(* IEC 61131-3 sources: elnaProjects/kc6/build_BaseProject_ecl/_ (part 3) *)

  StrAlg.status :=  SHL(BYTE_TO_DWORD(source_for_Status), 29)
  			OR SHL(BYTE_TO_DWORD(cmd_for_Status), 26)
  			OR SHL(BYTE_TO_DWORD(command_error_for_Status), 23)
  			OR SHL(BOOL_TO_DWORD(StrAlg.OpcCommandsDisabled ), 21)
  			OR SHL(BOOL_TO_DWORD(StrAlg.hasError),4)
  			OR SHL(BOOL_TO_DWORD(StrAlg.CanRun),2)
  			OR SHL(BOOL_TO_DWORD(StrAlg.isEnded),1)
  			OR BOOL_TO_DWORD(StrAlg.isRuning);
END_FUNCTION_BLOCK

FUNCTION_BLOCK TestProtectionAlg
  VAR_IN_OUT
    StrAlg : struct_Alg;
  END_VAR
  VAR
    _sunpackerCommand : fb_sunpackerCommand;
    source : BYTE;
    cmd : BYTE;
    lastCmd : BYTE;
    source_for_Status : BYTE;
    cmd_for_Status : BYTE;
    command_error_for_Status : BYTE;
    resetCmdTimer : TON;
    resetCmdTimerPriznak : BOOL;
  END_VAR
  VAR_EXTERNAL
    ai : AiConfig;
    protectManager : struct_ProtectionsManager;
    algManager : struct_AlgoritmsManager;
    ModeGpa : TYPE_ModeGpa;
    PMcommand : TYPE_CommandsPotectionsManager;
  END_VAR

  StrAlg.CanRun := StrAlg.inCanRun;
  StrAlg.OpcCommandsDisabled := StrAlg.inOpcCommandsDisabled;

  (* ---- Если управление с ВУ заблокировано, то передаем команду из алгоритма ---- *)
  IF StrAlg.inOpcCommandsDisabled THEN
  	StrAlg.inCommand := StrAlg.inCommand_Alg;
  ELSE (* иначе передаем команду с АРМа*)
  	StrAlg.inCommand := StrAlg.inCommand_ARM;
  END_IF;

  _sunpackerCommand(command := StrAlg.inCommand);
  	source := _sunpackerCommand.source;
  	cmd := _sunpackerCommand.cmd;

  IF cmd <> 0 AND lastCmd <> cmd AND (((NOT StrAlg.opcCommandsDisabled) AND source > 0) OR source = 0) then
  	CASE BYTE_TO_INT(cmd) OF
  		(*cmdRun*) 1: 	IF (StrAlg.CanRun) THEN
  					StrAlg.isRuning := TRUE;
  					StrAlg.isEnded := FALSE;
  					StrAlg.hasError 	:= FALSE;
                                               (*****************       OnRun       *****************)
                                                        algManager.nMode:=ModeGpa.MODE_TESTAZ;
                                                        protectManager.inCommand:=PMcommand.CheckProtections;
  					    EnableAiLimits(ai);
                                                    (*StrAlg.inOpcCommandsDisabled:=FALSE;*)
  					cmd_for_Status := cmd;
  					source_for_Status := source;
  					command_error_for_Status := 0;
  				ELSE
  					StrAlg.isRuning := FALSE;
  					StrAlg.isEnded := FALSE;
  					StrAlg.hasError 	:= FALSE;

  					cmd_for_Status := 0;
  					source_for_Status := source;
  					command_error_for_Status := cmd;
  				END_IF;
  		(*cmdReset*) 2: 	StrAlg.isRuning := FALSE;
  				StrAlg.isEnded := FALSE;
  				StrAlg.hasError 	:= FALSE;
                                          (*****************       OnReset       *****************)
                                                    DisableAiLimits(ai);
                                                    protectManager.inCommand:=PMcommand.RestartAllProtections;
                                                    algManager.nMode:=ModeGpa.MODE_STOP;

  				cmd_for_Status := cmd;
  				source_for_Status := source;
  				command_error_for_Status := 0;
  	END_CASE;
  	resetCmdTimer(IN := false);
  	resetCmdTimerPriznak := TRUE;
  END_IF;
  lastCmd := cmd;

  resetCmdTimer(IN := resetCmdTimerPriznak, PT := T#5S);
  IF resetCmdTimer.Q THEN
  	resetCmdTimerPriznak := FALSE;
  	source_for_Status := 0;
  	cmd_for_Status := 0;
  	command_error_for_Status := 0;
  END_IF;

  StrAlg.status :=  SHL(BYTE_TO_DWORD(source_for_Status), 29)
  			OR SHL(BYTE_TO_DWORD(cmd_for_Status), 26)
  			OR SHL(BYTE_TO_DWORD(command_error_for_Status), 23)
  			OR SHL(BOOL_TO_DWORD(StrAlg.OpcCommandsDisabled ), 21)
  			OR SHL(BOOL_TO_DWORD(StrAlg.hasError),4)
  			OR SHL(BOOL_TO_DWORD(StrAlg.CanRun),2)
  			OR SHL(BOOL_TO_DWORD(StrAlg.isEnded),1)
  			OR BOOL_TO_DWORD(StrAlg.isRuning);
END_FUNCTION_BLOCK

FUNCTION_BLOCK engineRunAlg
  VAR_IN_OUT
    StrAlg : struct_Alg;
  END_VAR
  VAR
    BreakPuskTimer : struct_PhaseAlgoritm;
    RunProtection_mvoff : struct_PhaseAlgoritm;
    LowOil_upStopust : struct_PhaseAlgoritm;
    mvOn : struct_PhaseAlgoritm;
    AutoPns_ph : struct_PhaseAlgoritm;
    AutoAvom_ph : struct_PhaseAlgoritm;
    pnsOff : struct_PhaseAlgoritm;
    testUnsuccessful : struct_PhaseAlgoritm;
    fb_BreakPuskTimer : fb_ph_Timer;
    fb_RunProtection_mvoff : fb_ph_DIprotection;
    fb_LowOil_upStopust : fb_ph_WaitAnalogValue;
    fb_mvOn : fb_ph_SectionSwitch;
    fb_AutoPns_ph : fb_ph_algoritm;
    fb_AutoAvom_ph : fb_ph_algoritm;
    fb_pnsOff : fb_ph_Switch;
    fb_testUnsuccessful : fb_ph_CustomPhase;
    _sunpackerCommand : fb_sunpackerCommand;
    _DualStateImAction : TYPE_DualStateImAction;
    _PhaseAlgoritmAction : TYPE_PhaseAlgoritmAction;
    source : BYTE;
    cmd : BYTE;
    lastCmd : BYTE;
    source_for_Status : BYTE;
    cmd_for_Status : BYTE;
    command_error_for_Status : BYTE;
    resetCmdTimer : TON;
    resetCmdTimerPriznak : BOOL;
    onInit : BOOL;
    waitReset : TON;
  END_VAR
  VAR_EXTERNAL
    IM : ImConfig;
    algoritms : AlgoritmsConfig;
    ai : AiConfig;
    protections : ProtectionsConfig;
    AlgTimers : struct_AlgTimers;
  END_VAR

  IF NOT onInit THEN

       fb_BreakPuskTimer(phaseNumber:=0, delay:=T#665S);
     fb_LowOil_upStopust(phaseNumber:=1);
                 fb_mvOn(phaseNumber:=2, act:=_on);
           fb_AutoPns_ph(phaseNumber:=3, act:=_run, waitCompletion:=FALSE);
          fb_AutoAvom_ph(phaseNumber:=4, act:=_run, waitCompletion:=FALSE);
               fb_pnsOff(phaseNumber:=5, act:=_off);
  fb_RunProtection_mvoff(phaseNumber:=7, act:=_run);
     fb_testUnsuccessful(phaseNumber:=17);

  onInit:=TRUE;
  END_IF;

          fb_BreakPuskTimer(StrPh:=BreakPuskTimer, timer:=AlgTimers.engineRun_BreakPuskTimer);
        fb_LowOil_upStopust(StrPh:=LowOil_upStopust, ai:=ai.Davlenie_masla_smazki_nizkoe, more:=im.AutoPns_UstStop.Value);
                    fb_mvOn(StrPh:=mvOn, Im:=Im.MB);
              fb_AutoPns_ph(StrPh:=AutoPns_ph, alg:=algoritms.AutoPns);
             fb_AutoAvom_ph(StrPh:=AutoAvom_ph, alg:=algoritms.AutoAvom);
                  fb_pnsOff(StrPh:=pnsOff, Im:=Im.pns);
     fb_RunProtection_mvoff(StrPh:=RunProtection_mvoff, StrDiP:=protections.MB);
        fb_testUnsuccessful(StrPh:=testUnsuccessful);

  StrAlg.CanRun := StrAlg.inCanRun;
  StrAlg.OpcCommandsDisabled := StrAlg.inOpcCommandsDisabled;

  IF StrAlg.isRuning THEN

      StrAlg.hasError := mvOn.error OR pnsOff.error OR testUnsuccessful.error;

      IF mvOn.top THEN
          runPhase(RunProtection_mvoff);
          runPhase(AutoAvom_ph);
          runPhase(LowOil_upStopust);
      END_IF;

      IF LowOil_upStopust.top THEN
          runPhase(pnsOff);
      END_IF;

      IF pnsOff.top THEN
         runPhase(AutoPns_ph);
      END_IF;

      IF BreakPuskTimer.top AND NOT AutoPns_ph.top THEN
            testUnsuccessful.error:=TRUE;
      END_IF;

      IF AutoPns_ph.top THEN
            resetPhase(BreakPuskTimer);
  	waitReset(IN:=TRUE, PT:= T#2S);
      END_IF;

      IF waitReset.Q AND NOT (algoritms.Apusk.isRuning OR algoritms.SemiAutoPusk.isRuning) THEN
  	resetIfRunning(StrAlg);
      END_IF;

      StrAlg.isEnded:= AutoPns_ph.top;
  END_IF;

  StrAlg.CanRun := StrAlg.inCanRun;
  StrAlg.OpcCommandsDisabled := StrAlg.inOpcCommandsDisabled;

  (* ---- Если управление с ВУ заблокировано, то  передаем команду из алгоритма ---- *)
  IF StrAlg.inOpcCommandsDisabled THEN
  	StrAlg.inCommand := StrAlg.inCommand_Alg;
  ELSE (* иначе передаем команду с АРМа*)
  	StrAlg.inCommand := StrAlg.inCommand_ARM;
  END_IF;

  _sunpackerCommand(command := StrAlg.inCommand);
  	source := _sunpackerCommand.source;
  	cmd := _sunpackerCommand.cmd;

  IF cmd <> 0 AND lastCmd <> cmd AND (((NOT StrAlg.opcCommandsDisabled) AND source > 0) OR source = 0) then
  	CASE BYTE_TO_INT(cmd) OF
  		(*cmdRun*) 1: 	IF (StrAlg.CanRun) THEN
  					StrAlg.isRuning := TRUE;
  					StrAlg.isEnded := FALSE;
  					StrAlg.hasError := FALSE;
  					(*****************       OnRun       *****************)

                                                    runPhase(mvOn);
                                                    runPhase(BreakPuskTimer);
                                                    runPhase(testUnsuccessful);

  					cmd_for_Status := cmd;
  					source_for_Status := source;
  					command_error_for_Status := 0;
  				ELSE
  					StrAlg.isRuning := FALSE;
  					StrAlg.isEnded := FALSE;
  					StrAlg.hasError 	:= FALSE;

  					cmd_for_Status := 0;
  					source_for_Status := source;
  					command_error_for_Status := cmd;
  				END_IF;
  		(*cmdReset*) 2: 	StrAlg.isRuning := FALSE;
  				StrAlg.isEnded := FALSE;
  				StrAlg.hasError 	:= FALSE;

                                           (*****************       OnReset       *****************)
                                          StrAlg.inCanRun:=FALSE;
                                          waitReset(IN:=FALSE);

                                          resetPhase(BreakPuskTimer);
                                          resetPhase(RunProtection_mvoff);
                                          resetPhase(LowOil_upStopust);
                                          resetPhase(mvOn);
                                          resetPhase(AutoPns_ph);
                                          resetPhase(AutoAvom_ph);
                                          resetPhase(pnsOff);
                                          resetPhase(testUnsuccessful);

  				cmd_for_Status := cmd;
  				source_for_Status := source;
  				command_error_for_Status := 0;
  	END_CASE;
  	resetCmdTimer(IN := false);
  	resetCmdTimerPriznak := TRUE;
  END_IF;
  lastCmd := cmd;

  resetCmdTimer(IN := resetCmdTimerPriznak, PT := T#5S);
  IF resetCmdTimer.Q THEN
  	resetCmdTimerPriznak := FALSE;
  	source_for_Status := 0;
  	cmd_for_Status := 0;
  	command_error_for_Status := 0;
  END_IF;

  StrAlg.Start:= BreakPuskTimer.startStatus
              OR RunProtection_mvoff.startStatus
              OR LowOil_upStopust.startStatus
              OR mvOn.startStatus
              OR AutoPns_ph.startStatus
              OR AutoAvom_ph.startStatus
              OR pnsOff.startStatus
              OR testUnsuccessful.startStatus;

  StrAlg.Error:= BreakPuskTimer.errorStatus
              OR RunProtection_mvoff.errorStatus
              OR LowOil_upStopust.errorStatus
              OR mvOn.errorStatus
              OR AutoPns_ph.errorStatus
              OR AutoAvom_ph.errorStatus
              OR pnsOff.errorStatus
              OR testUnsuccessful.errorStatus;

  StrAlg.Top:=   BreakPuskTimer.topStatus
              OR RunProtection_mvoff.topStatus
              OR LowOil_upStopust.topStatus
              OR mvOn.topStatus
              OR AutoPns_ph.topStatus
              OR AutoAvom_ph.topStatus
              OR pnsOff.topStatus
              OR testUnsuccessful.topStatus;

  (*TODO: TYPE PROGRAM CODE HERE*)
  StrAlg.status :=  SHL(BYTE_TO_DWORD(source_for_Status), 29)
  			OR SHL(BYTE_TO_DWORD(cmd_for_Status), 26)
  			OR SHL(BYTE_TO_DWORD(command_error_for_Status), 23)
  			OR SHL(BOOL_TO_DWORD(StrAlg.OpcCommandsDisabled ), 21)
  			OR SHL(BOOL_TO_DWORD(StrAlg.hasError),4)
  			OR SHL(BOOL_TO_DWORD(StrAlg.CanRun),2)
  			OR SHL(BOOL_TO_DWORD(StrAlg.isEnded),1)
  			OR BOOL_TO_DWORD(StrAlg.isRuning);
END_FUNCTION_BLOCK

FUNCTION_BLOCK fb_AI_Init
  VAR_INPUT
    data_Ini : BOOL;
    dLL : LREAL;
    dHL : LREAL;
    dLA : LREAL;
    dHA : LREAL;
    dLW : LREAL;
    dHW : LREAL;
    ISVALIDREF_LA : BOOL         := False;
    ISVALIDREF_HA : BOOL         := False;
    ISVALIDREF_LW : BOOL         := False;
    ISVALIDREF_HW : BOOL         := False;
    delayLA : TIME         := T#0S;
    delayLW : TIME         := T#0S;
    delayHW : TIME         := T#0S;
    delayHA : TIME         := T#0S;
    inpLL : LREAL         := 4000.0;
    inpHL : LREAL         := 20000.0;
    CurrentShotCircuit : LREAL         := 21000.0;
    CurrentBreakCircuit : LREAL         := 3700.0;
    dMaxChangeSpeed : LREAL;
    dMaxChangeSpeedDown : LREAL;
    histeresis : LREAL;
    aperturFilter : LREAL;
    exponentialFilter : LREAL;
    rassoglasovanie : LREAL;
    inOpcCommandsDisabled : BOOL;
  END_VAR
  VAR_IN_OUT
    strAI : struct_AI;
  END_VAR
  VAR_OUTPUT
    Init : BOOL         := FALSE;
  END_VAR

  (*****            Функциональный блок переинициализации структуры-дескриптора канала аналогового ввода.            *****)
       Init := false;

      IF data_Ini THEN                            (* Параметрам требуется переинициализация. *)
          strAI.dLL                := dLL;
          strAI.dHL                := dHL;
          strAI.dLA                := dLA;
          strAI.dHA                := dHA;
          strAI.dLW                := dLW;
          strAI.dHW                := dHW;
          strAI.ISVALIDREF_LA      := ISVALIDREF_LA;
          strAI.ISVALIDREF_HA      := ISVALIDREF_HA;
          strAI.ISVALIDREF_LW      := ISVALIDREF_LW;
          strAI.ISVALIDREF_HW      := ISVALIDREF_HW;
          strAI.delayLA            := delayLA;
          strAI.delayLW            := delayLW;
          strAI.delayHW            := delayHW;
          strAI.delayHA            := delayHA;
          strAI.inpLL              := inpLL;
          strAI.inpHL              := inpHL;
          strAI.CurrentShotCircuit := CurrentShotCircuit;
          strAI.CurrentBreakCircuit:= CurrentBreakCircuit;
          strAI.dMaxChangeSpeed     := dMaxChangeSpeed;
          strAI.dMaxChangeSpeedDown := dMaxChangeSpeedDown;
          strAI.histeresis         := histeresis;
          strAI.aperturFilter      := aperturFilter;
          strAI.exponentialFilter  := exponentialFilter;
          strAI.rassoglasovanie    := rassoglasovanie;
          strAI.rassoglasovanie    := rassoglasovanie;

          data_Ini:=false;
          Init := TRUE;
       END_IF;
    IF Init THEN
          dLL:= 0.0;
          dHL:= 0.0;
          dLA:= 0.0;
          dHA:= 0.0;
          dLW:= 0.0;
          dHW:= 0.0;
          inpLL:= 4000.0;
          inpHL:= 20000.0;
          CurrentShotCircuit:= 21000.0;
          CurrentBreakCircuit:= 3700.0;
          ISVALIDREF_LA:= false;
          ISVALIDREF_HA:= false;
          ISVALIDREF_LW:= false;
          ISVALIDREF_HW:= false;
          delayLA:= T#0S;
          delayLW:= T#0S;
          delayHW:= T#0S;
          delayHA:= T#0S;
          dMaxChangeSpeed:= 0.0;
          dMaxChangeSpeedDown:= 0.0;
          histeresis:= 0.0;
          aperturFilter:= 0.0;
          exponentialFilter:= 0.0;
          rassoglasovanie:= 0.0;
        END_IF;
END_FUNCTION_BLOCK

FUNCTION_BLOCK fb_AOSourceMlp
  VAR_IN_OUT
    OutCurrent : TDoubleData;
    strAO : struct_AO;
  END_VAR
  VAR_INPUT
    retainLL : LREAL;
    retainHL : LREAL;
  END_VAR
  VAR
    _sunpackerCommand : fb_sunpackerCommand;
    source : BYTE;
    source_for_Status : BYTE;
    cmd : BYTE;
    cmd_for_Status : BYTE;
    lastCmd : BYTE;
    command_error_for_Status : BYTE;
    resetCmdTimer : TON;
    resetCmdTimerPriznak : BOOL;
    secondTack : BOOL;
    inOpcCommandsDisabled : BOOL;
  END_VAR

  IF NOT secondTack THEN
            IF (strAO.newLL <> retainLL) AND (retainLL <> 0.0) THEN  strAO.LL := retainLL;
            ELSE strAO.LL:= strAO.newLL; END_IF;
  	IF (strAO.newHL <> retainHL) AND (retainHL <> 0.0) THEN  strAO.HL := retainHL;
            ELSE strAO.HL:= strAO.newHL; END_IF;

  	secondTack  := FALSE;
  END_IF;
  strAO.blConnect :=(UINT_TO_WORD(OutCurrent.wFlags) AND 16#0040) <> 0;
  strAO.OpcCommandsDisabled := inOpcCommandsDisabled;

  _sunpackerCommand(command := strAO.inCommand);
  	source := _sunpackerCommand.source;
  	cmd := _sunpackerCommand.cmd;

  IF cmd <> 0 AND lastCmd <> cmd and (((NOT strAO.opcCommandsDisabled) AND source > 0) OR source = 0) then
  	CASE BYTE_TO_INT(cmd) OF
  	(*cmd_ChangeValue*) 1 : 	IF ((NOT strAO.newLL_ISVALIDREF) OR (strAO.nValue >= strAO.LL)) AND
                                             ((NOT strAO.newHL_ISVALIDREF) OR (strAO.nValue <= strAO.HL) ) THEN
  					strAO.Value := strAO.nValue;
  				END_IF;
  	(*cmd_ChangeLimits*) 2 : 	strAO.LL := strAO.newLL; retainLL:= strAO.LL;
  				strAO.HL := strAO.newHL; retainHL:= strAO.HL;
  	END_CASE;
  	source_for_Status := source;
  	cmd_for_Status := cmd;
  	command_error_for_Status := 0;
  	resetCmdTimer(IN := FALSE);
  	resetCmdTimerPriznak := TRUE;
  END_IF;
  lastCmd := cmd;

  IF (strAO.HL <> strAO.LL) THEN
  	OutCurrent.dblValue := ((strAO.Value - strAO.LL) * (strAO.outHL-strAO.outLL)/(strAO.HL - strAO.LL )) + strAO.outLL;
  END_IF;

  resetCmdTimer(IN := resetCmdTimerPriznak, PT := T#5S);
  IF resetCmdTimer.Q THEN
  	resetCmdTimerPriznak := FALSE;
  	source_for_Status := 0;
  	cmd_for_Status := 0;
  	command_error_for_Status := 0;
  END_IF;

  strAO.status := SHL(BYTE_TO_DWORD(source_for_Status), 29)
  			OR SHL(BYTE_TO_DWORD(cmd_for_Status), 26)
  			OR SHL(BYTE_TO_DWORD(command_error_for_Status), 23)
  			OR SHL(BOOL_TO_DWORD(strAO.OpcCommandsDisabled ), 21);
END_FUNCTION_BLOCK

FUNCTION_BLOCK fb_AO_Init
  VAR_INPUT
    data_Ini : BOOL;
    outLL : LREAL         := 4000.0;
    outHL : LREAL         := 20000.0;
    newLL : LREAL;
    newHL : LREAL;
    newLL_ISVALIDREF : BOOL;
    newHL_ISVALIDREF : BOOL;
  END_VAR
  VAR_IN_OUT
    strAO : struct_AO;
  END_VAR
  VAR_OUTPUT
    Init : BOOL         := FALSE;
  END_VAR

  (*****            Функциональный блок переинициализации структуры-дескриптора канала аналогового ввода.            *****)

   Init := FALSE;

      IF data_Ini THEN                            (* Параметрам требуется переинициализация. *)
          strAO.outLL                := outLL;
          strAO.outHL                := outHL;
          strAO.newLL                := newLL;
          strAO.newHL                := newHL;
          strAO.newLL_ISVALIDREF     := newLL_ISVALIDREF;
          strAO.newHL_ISVALIDREF     := newHL_ISVALIDREF;
          data_Ini:=FALSE;
          Init := TRUE;
      END_IF;
   IF Init THEN
         (* outLL:=0.0;*)
         (* outHL:=0.0;*)
          newLL:=0.0;
          newHL:=0.0;
          newLL_ISVALIDREF:= FALSE;
          newHL_ISVALIDREF:= FALSE;
   END_IF;
END_FUNCTION_BLOCK

FUNCTION_BLOCK fb_AiProtection
  VAR_INPUT
    ai : struct_AI;
  END_VAR
  VAR_IN_OUT
    StrAIp : struct_AiProtection;
  END_VAR
  VAR
    _sunpackerCommand : fb_sunpackerCommand;
    _signalingTp : TOF;
    _statusAi : TYPE_StatusAi;
    source : BYTE;
    cmd : BYTE;
    lastCmd : BYTE;
    source_for_Status : BYTE;
    cmd_for_Status : BYTE;
    command_error_for_Status : BYTE;
    resetCmdTimer : TON;
    resetCmdTimerPriznak : BOOL;
    signalinTimer : TON;
    timer : TON;
    SignalingTrig : R_TRIG;
    SignalingFTrig : F_TRIG;
    SignalingAi : BOOL;
  END_VAR

  timer(IN :=(ai.interval=StrAIp.controlLimit) AND (ai.interval >= _statusAi.normal) AND StrAIp.isRunning, PT :=StrAIp.delay);
  SignalingTrig(CLK := timer.Q);
  IF SignalingTrig.Q THEN
  	SignalingAi := TRUE;
  END_IF;
  SignalingFTrig(CLK := timer.Q);
  IF SignalingFTrig.Q THEN
  	SignalingAi := FALSE;
  END_IF;

  StrAIp.Tag := StrAIp.inTag;
  StrAIp.RunOnStart := StrAIp.inRunOnStart;

  StrAIp.CanRun := StrAIp.inCanRun;

  StrAIp.OpcCommandsDisabled := StrAIp.inOpcCommandsDisabled;

  (* ---- Если управление с ВУ заблокировано, то передаем команду из алгоритма ---- *)
  IF StrAIp.inOpcCommandsDisabled THEN
  	StrAIp.inCommand := StrAIp.inCommand_Alg;
  ELSE (* иначе передаем команду с АРМа*)
  	StrAIp.inCommand := StrAIp.inCommand_ARM;
  END_IF;

  _sunpackerCommand(command := StrAIp.inCommand);
  	source := _sunpackerCommand.source;
  	cmd := _sunpackerCommand.cmd;

  IF cmd <> 0 AND lastCmd <> cmd AND (((NOT StrAIp.opcCommandsDisabled) AND source > 0) OR source = 0) then

  	CASE BYTE_TO_INT(cmd) OF
  		(*cmdRun*) 1: 	IF        NOT StrAIp.Remont THEN
  					StrAIp.isEnded := FALSE;
  					StrAIp.hasError 	:= FALSE;
  					StrAIp.isRunning := TRUE;

  					cmd_for_Status := cmd;
  					source_for_Status := source;
  					command_error_for_Status := 0;
  				ELSE
  					StrAIp.isRunning := FALSE;
  					StrAIp.isEnded := FALSE;
  					StrAIp.hasError 	:= FALSE;

  					cmd_for_Status := 0;
  					source_for_Status := source;
  					command_error_for_Status := cmd;
  				END_IF;
                                          StrAIp.inopcCommandsDisabled:=FALSE;

  		(*cmdReset*) 2: 	StrAIp.isRunning := FALSE;
  				StrAIp.isEnded := FALSE;
  				StrAIp.hasError 	:= FALSE;
  				SignalingAi := FALSE;
  				StrAIp.Check := FALSE;
                                          (*StrAIp.Remont := FALSE;*)
  				cmd_for_Status := cmd;
  				source_for_Status := source;
  				command_error_for_Status := 0;
                                          StrAIp.inopcCommandsDisabled:=FALSE;

  	(*cmd_setRemont*) 4 :	StrAIp.Remont := TRUE;
  				(*StrAIp.isRunning := FALSE;*)

  				cmd_for_Status := cmd;
  				source_for_Status := source;
  				command_error_for_Status := 0;
  	(*cmd_resetRemont*) 5 : 	(*IF (ai.interval=StrAIp.controlLimit) THEN
  					cmd_for_Status := 0;
  					source_for_Status := 0;
  					command_error_for_Status := cmd;
  				ELSE*)
  					StrAIp.Remont := FALSE;
  					(*StrAIp.isRunning := TRUE;*)

  					cmd_for_Status := cmd;
  					source_for_Status := source;
  					command_error_for_Status := 0;
  				(*END_IF;*)
  	(*cmd_setCheck*) 6 : 	StrAIp.Check := TRUE;

  				cmd_for_Status := cmd;
  				source_for_Status := source;
  				command_error_for_Status := 0;
  	END_CASE;
  	resetCmdTimer(IN := false);
  	resetCmdTimerPriznak := TRUE;
  END_IF;
  lastCmd := cmd;

  resetCmdTimer(IN := resetCmdTimerPriznak);
  IF resetCmdTimer.Q THEN
  	resetCmdTimerPriznak := FALSE;
  	source_for_Status := 0;
  	cmd_for_Status := 0;
  	command_error_for_Status := 0;
  END_IF;

  IF StrAIp.isRunning AND NOT StrAIp.Remont AND NOT StrAIp.Check THEN
  	StrAIp.Signaling := SignalingAi;
  	StrAIp.SignalingTP := _signalingTp.Q;
  ELSE
  	StrAIp.Signaling := 0;
  	StrAIp.SignalingTP := 0;
  END_IF;

  _signalingTp(in := StrAIp.Signaling, PT := T#1s);

  StrAIp.status :=  SHL(BYTE_TO_DWORD(source_for_Status), 29)
  			OR SHL(BYTE_TO_DWORD(cmd_for_Status), 26)
  			OR SHL(BYTE_TO_DWORD(command_error_for_Status), 23)
  			OR SHL(BOOL_TO_DWORD(StrAIp.OpcCommandsDisabled ), 21)
  			OR SHL(BOOL_TO_DWORD(StrAIp.Signaling), 16)
  			OR SHL(BOOL_TO_DWORD(StrAIp.RunOnStart ), 15)
  			OR SHL(BOOL_TO_DWORD(StrAIp.remont), 6)
  			OR SHL(BOOL_TO_DWORD(StrAIp.Check), 5)
  			OR SHL(BOOL_TO_DWORD(StrAIp.hasError), 4)
  			OR SHL(BOOL_TO_DWORD(StrAIp.SignalingTP), 3)
  			OR SHL(BOOL_TO_DWORD(StrAIp.CanRun), 2)
  			OR SHL(BOOL_TO_DWORD(StrAIp.isEnded), 1)
  			OR BOOL_TO_DWORD(StrAIp.isRunning);
END_FUNCTION_BLOCK

FUNCTION_BLOCK fb_AiSourceMlp
  VAR_INPUT
    arAIN : TItemAIN;
    err_mod : TItemDIN;
  END_VAR
  VAR_IN_OUT
    strAI : struct_AI;
  END_VAR
  VAR
    _statusAi : TYPE_StatusAi;
    _commandAnalog : TYPE_CommandAnalog;
    _sunpackerCommand : fb_sunpackerCommand;
    _AnalogLimitFlags : TYPE_AnalogLimitFlags;
    notReliable : BOOL;
    _lastValue : LREAL;
    resetCmdTimer : TON;
    _LastValueTimer : TON;
    resetCmdTimerPriznak : BOOL;
    k : LREAL;
    b : LREAL;
    ap : LREAL;
    raznitsa : LREAL;
    rABS : LREAL;
    h : LREAL;
    mismatch : LREAL;
    parametr : BYTE;
    source : BYTE;
    cmd : BYTE;
    lastCmd : BYTE;
    source_for_Status : BYTE;
    cmd_for_Status : BYTE;
    command_error_for_Status : BYTE;
    onInit : BOOL;
    off_trig : R_TRIG;
    on_trig : R_TRIG;
    remont_trig : R_TRIG;
    LL_trig : R_TRIG;
    HL_trig : R_TRIG;
    Normal_trig : R_TRIG;
    Nedostover_trig : R_TRIG;
  END_VAR

  strAI.opcCommandsDisabled := strAI.inopcCommandsDisabled ;

  (* ---- При первом пуске принимаем значение уставок ---- *)
  IF NOT onInit THEN

            strAI.LL := strAI.dLL;
            strAI.HL := strAI.dHL;

            strAI.MaxChangeSpeed     := strAI.dMaxChangeSpeed;
            strAI.MaxChangeSpeedDown := strAI.dMaxChangeSpeedDown;

            IF strAI.ISVALIDREF_HA THEN strAI.HA := strAI.dHA; END_IF;

            IF strAI.ISVALIDREF_LA THEN strAI.LA := strAI.dLA; END_IF;

            IF strAI.ISVALIDREF_HW THEN strAI.HW := strAI.dHW; END_IF;

            IF strAI.ISVALIDREF_LW THEN strAI.LW := strAI.dLW; END_IF;

  	onInit  := TRUE;
  END_IF;

  (* ---- пересчет тока в физ величину ---- *)
  k := (strAI.HL - strAI.LL)/(strAI.inpHl - strAI.inpLL);
  b := strAI.LL - k * strAI.inpLL;
  strAI.value := k * arAIN.dblValue + b;

  (* ---- определение обрыва и кз ----- *)

  strAI.blConnect :=TRUE;(*(UINT_TO_WORD(arAIN.wFlags) = 1472) and (UINT_TO_WORD(err_mod.wValue) = 20) and (UINT_TO_WORD(err_mod.wFlags) = 192);*)
  IF NOT strAI.blConnect THEN
      strAI.interval := _statusAi.NOTDEFINED;
  ELSIF ((arAIN.dblValue < strAI.currentBreakCircuit) AND (strAI.currentBreakCircuit > 0.0)) OR ((strAI.interval = _statusAi.LL) AND (arAIN.dblValue < (strAI.currentBreakCircuit + 100.0))) THEN
      strAI.interval := _statusAi.LL;
  ELSIF ((arAIN.dblValue > strAI.currentShotCircuit) AND (strAI.currentShotCircuit > 0.0)) OR ((strAI.interval = _statusAi.HL) AND (arAIN.dblValue > (strAI.currentShotCircuit - 100.0))) THEN
      strAI.interval := _statusAi.HL;
  ELSE
      strAI.interval := _statusAi.normal;
  END_IF;

  IF NOT strAI.imit THEN
  	(* Расчет апертурного фильтра*)
  	ap := strAI.aperturFilter * 0.01 * (strAI.HL - strAI.LL);
  	IF strAI.aperturFilter <> 0.0 THEN raznitsa := strAI.value- _lastValue;
  		IF 	raznitsa < 0.0 	THEN 	rABS := -raznitsa; 		ELSE 	rABS := raznitsa; 		END_IF;
  		IF 	rABS > ap 	THEN 	strAI.value := strAI.value;	ELSE 	strAI.value := _lastValue; 	END_IF;
  	END_IF;

  	(* Расчет экпоненциального фильтра*)
  	IF strAI.exponentialFilter <> 0.0 THEN strAI.value := (strAI.exponentialFilter * strAI.value) + ((1.0 - strAI.exponentialFilter) * _lastValue); END_IF;
  ELSE
  	strAI.interval := _statusAi.normal;
  END_IF;

  IF notReliable THEN strAI.interval := _statusAi.NOTRELIABLE; END_IF;

  IF NOT notReliable THEN
  	IF strAI.interval >= _statusAi.normal THEN
  		strAI.interval := _statusAi.NOTDEFINED;
  		h := strAI.histeresis* 0.01 * (strAI.HL-strAI.LL);
  		(*определение выхода за аппаратные границы вынесено в GetData.здесь только для нужд имитации*)
  		IF strAI.imit THEN
  			mismatch := strAI.rassoglasovanie * 0.01 * (strAI.HL - strAI.LL);
  			IF ( strAI.value < strAI.LL - mismatch)   THEN strAI.interval := _statusAi.LL;
  			ELSIF  (strAI.value > strAI.Hl + mismatch) THEN strAI.interval := _statusAi.HL; END_IF;
  		ELSE
  			strAI.interval := _statusAi.normal;
  			IF strAI.ISVALIDREF_LA AND NOT strAI.Disabled_LA AND (strAI.interval = _statusAi.normal) THEN
  				IF (strAI.value  < strAI.LA) OR ((strAI.interval = _statusAi.LA)  AND ((strAI.value - h) < strAI.LA))  THEN
  					strAI.interval := _statusAi.LA;
  				END_IF;
  			END_IF;
  			IF strAI.ISVALIDREF_HA  AND NOT strAI.Disabled_HA AND (strAI.interval = _statusAi.normal)  THEN
  				IF (strAI.value > strAI.HA) OR ((strAI.interval = _statusAi.HA)  AND ((strAI.value + h) > strAI.HA))  THEN
  					strAI.interval := _statusAi.HA;
  				END_IF;
  			END_IF;
  			IF strAI.ISVALIDREF_LW AND NOT strAI.Disabled_LW AND (strAI.interval = _statusAi.normal)  THEN
  				IF (strAI.value < strAI.LW) OR ((strAI.interval = _statusAi.LW)  AND ((strAI.value - h) < strAI.LW)) THEN
  					strAI.interval := _statusAi.LW;
  				END_IF;
  			END_IF;
  			IF strAI.ISVALIDREF_HW AND NOT strAI.Disabled_HW  AND (strAI.interval = _statusAi.normal) THEN
  				IF (strAI.value > strAI.HW)  OR ((strAI.interval = _statusAi.HW)  AND ((strAI.value + h) > strAI.HW))   THEN
  					strAI.interval := _statusAi.HW;
  				END_IF;
  			END_IF;
  		END_IF;
  	END_IF;
  ELSE
  	strAI.interval := _statusAi.NOTRELIABLE;
  END_IF;

  IF strAI.remont THEN strAI.interval := _statusAi.NOTDEFINED; END_IF;

  (* ---- Если управление с ВУ заблокировано, то  передаем команду из алгоритма ---- *)
  IF strAI.inOpcCommandsDisabled THEN
  	strAI.inCommand := strAI.inCommand_Alg;
  ELSE (* иначе передаем команду с АРМа*)
  	strAI.inCommand := strAI.inCommand_ARM;
  END_IF;

  _sunpackerCommand(command := strAI.inCommand);
  	source := _sunpackerCommand.source;
  	parametr := _sunpackerCommand.parametr;
  	cmd := _sunpackerCommand.cmd;

  IF cmd <> 0 AND lastCmd <> cmd and (((NOT strAI.opcCommandsDisabled) AND source > 0) OR source = 0) then
  	CASE BYTE_TO_INT(cmd) OF
  	(*cmd_SetUstavki*) 1 :
  				IF ((parametr AND _AnalogLimitFlags.LL) <> 0)		             	THEN 	strAI.LL := strAI.dLL; END_IF;
  				IF ((parametr AND _AnalogLimitFlags.HL) <> 0)		 	          THEN	strAI.HL := strAI.dHL; END_IF;
  				IF ((parametr AND _AnalogLimitFlags.LA) <> 0) AND strAI.ISVALIDREF_LA 	THEN	strAI.LA := strAI.dLA; END_IF;
  				IF ((parametr AND _AnalogLimitFlags.HA) <> 0) AND strAI.ISVALIDREF_HA 	THEN	strAI.HA := strAI.dHA; END_IF;
  				IF ((parametr AND _AnalogLimitFlags.LW) <> 0) AND strAI.ISVALIDREF_LW 	THEN	strAI.LW := strAI.dLW; END_IF;
  				IF ((parametr AND _AnalogLimitFlags.HW) <> 0) AND strAI.ISVALIDREF_HW 	THEN	strAI.HW := strAI.dHW; END_IF;
                                          IF ((parametr AND _AnalogLimitFlags.SipUP)   <> 0) THEN    strAI.MaxChangeSpeed:=         strAI.dMaxChangeSpeed; END_IF;
  				IF ((parametr AND _AnalogLimitFlags.SipDown) <> 0) THEN    strAI.MaxChangeSpeedDown:= strAI.dMaxChangeSpeedDown; END_IF;

  	(*cmd_SetRemont*) 6 :
  				strAI.remont := TRUE;
  	(*cmd_ResetRemont*) 7 :
  				strAI.remont := FALSE;
  	(*cmd_kvitNotReliable*) 4 :
  				notReliable := FALSE;
  	END_CASE;
  	source_for_Status := source;
  	cmd_for_Status := cmd;
  	command_error_for_Status := 0;
  	resetCmdTimer(IN := FALSE);
  	resetCmdTimerPriznak := TRUE;
  END_IF;
  lastCmd := cmd;

  resetCmdTimer(IN := resetCmdTimerPriznak, PT := T#5S);
  IF resetCmdTimer.Q THEN
  	resetCmdTimerPriznak := FALSE;
  	source_for_Status := 0;
  	cmd_for_Status := 0;
  	command_error_for_Status := 0;
  END_IF;

  strAI.NS_Min := (strAI.value < strAI.minValue) AND strAI.minValue_ISVALIDREF;
  strAI.NS_Max := (strAI.value > strAI.maxValue) AND strAI.maxValue_ISVALIDREF;

  strAI.NS := (strAI.interval <= _statusAi.normal) AND NOT strAI.remont;

  Normal_trig(CLK := strAI.interval >= _statusAi.normal);

  IF NOT Normal_trig.Q THEN
  	_LastValueTimer(PT := T#1S);
  	IF (strAI.value<>_lastValue) OR _LastValueTimer.Q THEN
  		IF (_LastValueTimer.ET>T#0MS) THEN
  			strAI.ChangeSpeed:=(strAI.value-_lastValue)/(TIME_TO_LREAL(_LastValueTimer.ET)/1000.0);
  		END_IF;
  		_LastValueTimer(IN:=FALSE);

  		_LastValueTimer(IN:=TRUE);
  	END_IF;
  END_IF;
  _lastValue := strAI.value;

  IF ((strAI.maxChangeSpeed<>0.0) OR  (strAI.maxChangeSpeedDown<>0.0)) AND ( strAI.interval>=_statusAi.normal) THEN
  		IF (strAI.ChangeSpeed>0.0) THEN
  		    IF (strAI.ChangeSpeed > strAI.maxChangeSpeed) AND (strAI.maxChangeSpeed>0.0000001) THEN
  			 notReliable:=TRUE;
  		    END_IF;
  		ELSE
  		    IF (ABS(strAI.ChangeSpeed)>strAI.maxChangeSpeedDown) AND (strAI.maxChangeSpeedDown>0.0000001)  THEN
                                 notReliable:=TRUE;
  		    END_IF;
  		END_IF;

  END_IF;

  strAI.status := SHL(BYTE_TO_DWORD(source_for_Status), 29) 		              (* Источник команды *)
  			OR SHL(BYTE_TO_DWORD(cmd_for_Status), 26) 	    (* Команда *)
  			OR SHL(BYTE_TO_DWORD(command_error_for_Status), 23)   (* Ошибка команды *)
  			OR SHL(BOOL_TO_DWORD(strAI.OpcCommandsDisabled ), 21) (* Управление в ВУ заблокировано *)
  			OR SHL(BOOL_TO_DWORD(strAI.Disabled_HA), 9)		    (* ВА исключена из формирования интервала *)
  			OR SHL(BOOL_TO_DWORD(strAI.Disabled_LA), 8)		    (* НА исключена из формирования интервала *)
  			OR SHL(BOOL_TO_DWORD(strAI.Disabled_HW), 7)		    (* ВП исключена из формирования интервала *)
  			OR SHL(BOOL_TO_DWORD(strAI.Disabled_LW), 6)	              (* НП исключена из формирования интервала *)
  			OR SHL(BOOL_TO_DWORD(strAI.NS), 5)			    (* неиспарвность сигнала *)
  			OR SHL(BOOL_TO_DWORD(strAI.remont), 4)	              (* Выведен в ремонт *)
  			OR BYTE_TO_DWORD(strAI.interval);	              (* интервал *)
END_FUNCTION_BLOCK

FUNCTION_BLOCK fb_AiSourceMlp_timer
  VAR_INPUT
    arAIN : TItemAIN;
    err_mod : TItemDIN;
  END_VAR
  VAR_IN_OUT
    strAI : struct_AI;
  END_VAR
  VAR
    retainLL : LREAL;
    retainHL : LREAL;
    retainLA : LREAL;
    retainHA : LREAL;
    retainLW : LREAL;
    retainHW : LREAL;
    _statusAi : TYPE_StatusAi;
    _commandAnalog : TYPE_CommandAnalog;
    _sunpackerCommand : fb_sunpackerCommand;
    _AnalogLimitFlags : TYPE_AnalogLimitFlags;
    notReliable : BOOL;
    _lastValue : LREAL;
    resetCmdTimer : TON;
    _LastValueTimer : TON;
    resetCmdTimerPriznak : BOOL;
    k : LREAL;
    b : LREAL;
    ap : LREAL;
    raznitsa : LREAL;
    rABS : LREAL;
    h : LREAL;
    mismatch : LREAL;
    parametr : BYTE;
    source : BYTE;
    cmd : BYTE;
    lastCmd : BYTE;
    source_for_Status : BYTE;
    cmd_for_Status : BYTE;
    command_error_for_Status : BYTE;
    secondTakt : BOOL;
    off_trig : R_TRIG;
    on_trig : R_TRIG;
    remont_trig : R_TRIG;
    LL_trig : R_TRIG;
    HL_trig : R_TRIG;
    Normal_trig : R_TRIG;
    Nedostover_trig : R_TRIG;
    timerLA : TON;
    timerHA : TON;
    timerLW : TON;
    timerHW : TON;
  END_VAR

  strAI.opcCommandsDisabled := strAI.inopcCommandsDisabled ;

  (* ---- При первом пуске принимаем значение уставок ---- *)
  IF NOT secondTakt THEN
            IF (strAI.dLL <> retainLL) AND (retainLL <> 0.0) THEN  strAI.LL := retainLL;
            ELSE strAI.LL := strAI.dLL; END_IF;
  	IF (strAI.dHL <> retainHL) AND (retainHL <> 0.0) THEN  strAI.HL := retainHL;
            ELSE strAI.HL := strAI.dHL; END_IF;

            IF strAI.ISVALIDREF_HA AND (strAI.dHA <> retainHA) AND (retainHA <> 0.0) THEN  strAI.HA := retainHA;
            ELSE strAI.HA := strAI.dHA; END_IF;

            IF strAI.ISVALIDREF_LA AND (strAI.dLA <> retainLA) AND (retainLA <> 0.0) THEN  strAI.LA := retainLA;
            ELSE strAI.LA := strAI.dLA; END_IF;

            IF strAI.ISVALIDREF_HW AND (strAI.dHW <> retainHW) AND (retainHW <> 0.0) THEN  strAI.HW := retainHW;
            ELSE strAI.HW := strAI.dHW; END_IF;

            IF strAI.ISVALIDREF_LW AND (strAI.dLW <> retainLW) AND (retainLW <> 0.0) THEN  strAI.LW := retainLW;
            ELSE strAI.LW := strAI.dLW; END_IF;

  	secondTakt  := TRUE;
  END_IF;

  (* ---- пересчет тока в физ величину ---- *)
  k := (strAI.HL - strAI.LL)/(strAI.inpHl - strAI.inpLL);
  b := strAI.LL - k * strAI.inpLL;
  strAI.value := k * arAIN.dblValue + b;

  (* ---- определение обрыва и кз ----- *)

  strAI.blConnect := true;(*(UINT_TO_WORD(arAIN.wFlags) = 1472) and (UINT_TO_WORD(err_mod.wValue) = 20) and (UINT_TO_WORD(err_mod.wFlags) = 192); *)
  IF NOT strAI.blConnect THEN
      strAI.interval := _statusAi.NOTDEFINED;
  ELSIF ((arAIN.dblValue < strAI.currentBreakCircuit) AND (strAI.currentBreakCircuit > 0.0)) OR ((strAI.interval = _statusAi.LL) AND (arAIN.dblValue < (strAI.currentBreakCircuit + 100.0))) THEN
      strAI.interval := _statusAi.LL;
  ELSIF ((arAIN.dblValue > strAI.currentShotCircuit) AND (strAI.currentShotCircuit > 0.0)) OR ((strAI.interval = _statusAi.HL) AND (arAIN.dblValue > (strAI.currentShotCircuit - 100.0))) THEN
      strAI.interval := _statusAi.HL;
  ELSE
      strAI.interval := _statusAi.normal;
  END_IF;

  IF NOT strAI.imit THEN
  	(* Расчет апертурного фильтра*)
  	ap := strAI.aperturFilter * 0.01 * (strAI.HL - strAI.LL);
  	IF strAI.aperturFilter <> 0.0 THEN raznitsa := strAI.value- _lastValue;
  		IF 	raznitsa < 0.0 	THEN 	rABS := -raznitsa; 		ELSE 	rABS := raznitsa; 		END_IF;
  		IF 	rABS > ap 	THEN 	strAI.value := strAI.value;	ELSE 	strAI.value := _lastValue; 	END_IF;
  	END_IF;

  	(* Расчет экпоненциального фильтра*)
  	IF strAI.exponentialFilter <> 0.0 THEN strAI.value := (strAI.exponentialFilter * strAI.value) + ((1.0 - strAI.exponentialFilter) * _lastValue); END_IF;
  ELSE
  	strAI.interval := _statusAi.normal;
  END_IF;

  IF notReliable THEN strAI.interval := _statusAi.NOTRELIABLE; END_IF;

  IF NOT notReliable THEN
  	IF strAI.interval >= _statusAi.normal THEN
  		strAI.interval := _statusAi.NOTDEFINED;
  		h := strAI.histeresis* 0.01 * (strAI.HL-strAI.LL);
  		(*определение выхода за аппаратные границы вынесено в GetData.здесь только для нужд имитации*)
  		IF strAI.imit THEN
  			mismatch := strAI.rassoglasovanie * 0.01 * (strAI.HL - strAI.LL);
  			IF ( strAI.value < strAI.LL - mismatch)   THEN strAI.interval := _statusAi.LL;
  			ELSIF  (strAI.value > strAI.Hl + mismatch) THEN strAI.interval := _statusAi.HL; END_IF;
  		ELSE
  			strAI.interval := _statusAi.normal;
  			IF strAI.ISVALIDREF_LA AND NOT strAI.Disabled_LA AND (strAI.interval = _statusAi.normal) THEN
                                timerLA(IN:=(strAI.value  < strAI.LA) OR ((strAI.interval = _statusAi.LA)  AND ((strAI.value - h) < strAI.LA)), PT:=strAI.delayLA);
  				IF timerLA.Q  THEN
  					strAI.interval := _statusAi.LA;
  				END_IF;
  			END_IF;
  			IF strAI.ISVALIDREF_HA  AND NOT strAI.Disabled_HA AND (strAI.interval = _statusAi.normal)  THEN
                                timerHA(IN:=(strAI.value > strAI.HA) OR ((strAI.interval = _statusAi.HA)  AND ((strAI.value + h) > strAI.HA)), PT:=strAI.delayHA);
  				IF timerHA.Q  THEN
  					strAI.interval := _statusAi.HA;
  				END_IF;
  			END_IF;
  			IF strAI.ISVALIDREF_LW AND NOT strAI.Disabled_LW AND (strAI.interval = _statusAi.normal)  THEN
                                timerLW(IN:=(strAI.value < strAI.LW) OR ((strAI.interval = _statusAi.LW)  AND ((strAI.value - h) < strAI.LW)), PT:=strAI.delayLW);
  				IF timerLW.Q THEN
  					strAI.interval := _statusAi.LW;
  				END_IF;
  			END_IF;
  			IF strAI.ISVALIDREF_HW AND NOT strAI.Disabled_HW  AND (strAI.interval = _statusAi.normal) THEN
                                timerHW(IN:=(strAI.value > strAI.HW)  OR ((strAI.interval = _statusAi.HW)  AND ((strAI.value + h) > strAI.HW)), PT:=strAI.delayHW);
  				IF  timerHW.Q  THEN
  					strAI.interval := _statusAi.HW;
  				END_IF;
  			END_IF;
  		END_IF;
  	END_IF;
  ELSE
  	strAI.interval := _statusAi.NOTRELIABLE;
  END_IF;

  IF strAI.remont THEN strAI.interval := _statusAi.NOTDEFINED; END_IF;

  _sunpackerCommand(command := strAI.inCommand);
  	source := _sunpackerCommand.source;
  	parametr := _sunpackerCommand.parametr;
  	cmd := _sunpackerCommand.cmd;

  IF cmd <> 0 AND lastCmd <> cmd and (((NOT strAI.opcCommandsDisabled) AND source > 0) OR source = 0) then
  	CASE BYTE_TO_INT(cmd) OF
  	(*cmd_SetUstavki*) 1 :
  				IF ((parametr AND _AnalogLimitFlags.LL) <> 0)		             	THEN 	strAI.LL := strAI.dLL; retainLL:= strAI.LL; END_IF;
  				IF ((parametr AND _AnalogLimitFlags.HL) <> 0)		 	          THEN	strAI.HL := strAI.dHL; retainHL:= strAI.HL; END_IF;
  				IF ((parametr AND _AnalogLimitFlags.LA) <> 0) AND strAI.ISVALIDREF_LA 	THEN	strAI.LA := strAI.dLA; retainLA:= strAI.LA; END_IF;
  				IF ((parametr AND _AnalogLimitFlags.HA) <> 0) AND strAI.ISVALIDREF_HA 	THEN	strAI.HA := strAI.dHA; retainHA:= strAI.HA; END_IF;
  				IF ((parametr AND _AnalogLimitFlags.LW) <> 0) AND strAI.ISVALIDREF_LW 	THEN	strAI.LW := strAI.dLW; retainLW:= strAI.LW; END_IF;
  				IF ((parametr AND _AnalogLimitFlags.HW) <> 0) AND strAI.ISVALIDREF_HW 	THEN	strAI.HW := strAI.dHW; retainHW:= strAI.HW; END_IF;
  	(*cmd_SetRemont*) 2 :
  				strAI.remont := TRUE;
  	(*cmd_ResetRemont*) 3 :
  				strAI.remont := FALSE;
  	(*cmd_kvitNotReliable*) 4 :
  				notReliable := FALSE;
  	END_CASE;
  	source_for_Status := source;
  	cmd_for_Status := cmd;
  	command_error_for_Status := 0;
  	resetCmdTimer(IN := FALSE);
  	resetCmdTimerPriznak := TRUE;
  END_IF;
  lastCmd := cmd;

  resetCmdTimer(IN := resetCmdTimerPriznak, PT := T#5S);
  IF resetCmdTimer.Q THEN
  	resetCmdTimerPriznak := FALSE;
  	source_for_Status := 0;
  	cmd_for_Status := 0;
  	command_error_for_Status := 0;
  END_IF;

  strAI.NS_Min := (strAI.value < strAI.minValue) AND strAI.minValue_ISVALIDREF;
  strAI.NS_Max := (strAI.value > strAI.maxValue) AND strAI.maxValue_ISVALIDREF;

  strAI.NS := (strAI.interval <= _statusAi.normal) AND NOT strAI.remont;

  Normal_trig(CLK := strAI.interval >= _statusAi.normal);

  IF NOT Normal_trig.Q THEN
  	_LastValueTimer(PT := T#1S);
  	IF (strAI.value<>_lastValue) OR _LastValueTimer.Q THEN
  		IF (_LastValueTimer.ET>T#0MS) THEN
  			strAI.ChangeSpeed:=(strAI.value-_lastValue)/(TIME_TO_LREAL(_LastValueTimer.ET)/1000.0);
  		END_IF;
  		_LastValueTimer(IN:=FALSE);

  		_LastValueTimer(IN:=TRUE);
  	END_IF;
  END_IF;
  _lastValue := strAI.value;

  IF ((strAI.maxChangeSpeed<>0.0) OR  (strAI.maxChangeSpeedDown<>0.0)) AND ( strAI.interval>=_statusAi.normal) THEN
  		IF (strAI.ChangeSpeed>0.0) THEN
  		    IF (strAI.ChangeSpeed > strAI.maxChangeSpeed) AND (strAI.maxChangeSpeed>0.0000001) THEN
  			 notReliable:=TRUE;
  		    END_IF;
  		ELSE
  		    IF (ABS(strAI.ChangeSpeed)>strAI.maxChangeSpeedDown) AND (strAI.maxChangeSpeedDown>0.0000001)  THEN
                                 notReliable:=TRUE;
  		    END_IF;
  		END_IF;

  END_IF;

  strAI.status := SHL(BYTE_TO_DWORD(source_for_Status), 29) 		              (* Источник команды *)
  			OR SHL(BYTE_TO_DWORD(cmd_for_Status), 26) 	    (* Команда *)
  			OR SHL(BYTE_TO_DWORD(command_error_for_Status), 23)   (* Ошибка команды *)
  			OR SHL(BOOL_TO_DWORD(strAI.OpcCommandsDisabled ), 21) (* Управление в ВУ заблокировано *)
  			OR SHL(BOOL_TO_DWORD(strAI.Disabled_HA), 9)		    (* ВА исключена из формирования интервала *)
  			OR SHL(BOOL_TO_DWORD(strAI.Disabled_LA), 8)		    (* НА исключена из формирования интервала *)
  			OR SHL(BOOL_TO_DWORD(strAI.Disabled_HW), 7)		    (* ВП исключена из формирования интервала *)
  			OR SHL(BOOL_TO_DWORD(strAI.Disabled_LW), 6)	              (* НП исключена из формирования интервала *)
  			OR SHL(BOOL_TO_DWORD(strAI.NS), 5)			    (* неиспарвность сигнала *)
  			OR SHL(BOOL_TO_DWORD(strAI.remont), 4)	              (* Выведен в ремонт *)
  			OR BYTE_TO_DWORD(strAI.interval);	              (* интервал *)
END_FUNCTION_BLOCK

FUNCTION_BLOCK fb_AnalogParametr
  VAR_IN_OUT
    StrAP : struct_AnalogParametr;
  END_VAR
  VAR
    _sunpackerCommand : fb_sunpackerCommand;
    source : BYTE;
    cmd : BYTE;
    source_for_Status : BYTE;
    cmd_for_Status : BYTE;
    command_error_for_Status : BYTE;
    resetCmdTimer : TON;
    resetCmdTimerPriznak : BOOL;
    secondTact : BOOL;
    inp : LREAL;
    rABS : LREAL;
  END_VAR

  IF NOT secondTact THEN
  	StrAP.Value := StrAP.currentValue;
  	secondTact := true;
  END_IF;

  StrAP.OpcCommandsDisabled := StrAP.inOpcCommandsDisabled;

   (* ---- Если управление с ВУ заблокировано, то передаем команду из алгоритма ---- *)
  IF StrAP.inOpcCommandsDisabled THEN
  	StrAP.inCommand := StrAP.inCommand_Alg;
  ELSE (* иначе передаем команду с АРМа*)
  	StrAP.inCommand := StrAP.inCommand_ARM;
  END_IF;

  _sunpackerCommand(command := StrAP.inCommand);
  	source := _sunpackerCommand.source;
  	cmd := _sunpackerCommand.cmd;

  IF cmd <> 0 AND StrAP.newValue <> StrAP.Value and (((NOT StrAP.opcCommandsDisabled) AND source > 0) OR source = 0) then
  	CASE BYTE_TO_INT(cmd) OF
  	(*cmd_ChangeValue*) 1 :
  				StrAP.isValidValue := TRUE;
  				IF StrAP.minVal_ISVALIDREF AND StrAP.isValidValue THEN
  					IF StrAP.newValue < StrAP.minVal THEN
  						StrAP.isValidValue := FALSE;
  					END_IF;
  				END_IF;
  				IF StrAP.maxVal_ISVALIDREF AND StrAP.isValidValue THEN
  					IF StrAP.newValue > StrAP.maxVal THEN
  						StrAP.isValidValue := FALSE;
  					END_IF;
  				END_IF;
  				IF StrAP.maxStep_ISVALIDREF AND StrAP.isValidValue  THEN
  					inp := StrAP.Value - StrAP.newValue;
  					IF inp < 0.0 THEN
  						rABS := -inp;
  					ELSE
  						rABS := inp;
  					END_IF;
  					IF rABS > StrAP.maxStep THEN
  						StrAP.isValidValue := FALSE;
  					END_IF;
  				END_IF;
  				IF StrAP.isValidValue THEN
  					StrAP.Value := StrAP.newValue;
  					command_error_for_Status := 0;
  				ELSE
  					command_error_for_Status := cmd;
  				END_IF;
  	END_CASE;
  	source_for_Status := source;
  	cmd_for_Status := cmd;
  	resetCmdTimer(IN := FALSE);
  	resetCmdTimerPriznak := TRUE;
  END_IF;

  resetCmdTimer(IN := resetCmdTimerPriznak, PT := T#5S);
  IF resetCmdTimer.Q THEN
  	resetCmdTimerPriznak := FALSE;
  	source_for_Status := 0;
  	cmd_for_Status := 0;
  	command_error_for_Status := 0;
  END_IF;

  StrAP.status := SHL(BYTE_TO_DWORD(source_for_Status), 29)
  			OR SHL(BYTE_TO_DWORD(cmd_for_Status), 26)
  			OR SHL(BYTE_TO_DWORD(command_error_for_Status), 23)
  			OR SHL(BOOL_TO_DWORD(StrAP.OpcCommandsDisabled ), 21);
END_FUNCTION_BLOCK

FUNCTION_BLOCK fb_AnalogParametr_Init
  VAR_INPUT
    data_Ini : BOOL;
    currentValue : LREAL;
    minVal : LREAL;
    maxVal : LREAL;
    maxStep : LREAL;
    minVal_ISVALIDREF : BOOL;
    maxVal_ISVALIDREF : BOOL;
    maxStep_ISVALIDREF : BOOL;
  END_VAR
  VAR_IN_OUT
    strAP : struct_AnalogParametr;
  END_VAR
  VAR_OUTPUT
    Init : BOOL         := FALSE;
  END_VAR

  (*****            Функциональный блок переинициализации Аналогового параметра.            *****)
       Init := false;

      IF data_Ini THEN                            (* Параметрам требуется переинициализация. *)
          strAP.currentValue          := currentValue;
          strAP.minVal                := minVal;
          strAP.maxVal                := maxVal;
          strAP.maxStep               := maxStep;
          strAP.minVal_ISVALIDREF     := minVal_ISVALIDREF;
          strAP.maxVal_ISVALIDREF     := maxVal_ISVALIDREF;
          strAP.maxStep_ISVALIDREF    := maxStep_ISVALIDREF;

          data_Ini:=false;
          Init := TRUE;
       END_IF;
       IF Init THEN
          currentValue:= 0.0;
          minVal:= 0.0;
          maxVal:= 0.0;
          maxStep:= 0.0;
          minVal_ISVALIDREF:= false;
          maxVal_ISVALIDREF:= false;
          maxStep_ISVALIDREF:= false;
       END_IF;
END_FUNCTION_BLOCK

FUNCTION_BLOCK fb_AutoAvomAlg
  VAR_IN_OUT
    StrAlg : struct_Alg;
    im1 : struct_Switch;
    im2 : struct_Switch;
  END_VAR
  VAR_INPUT
    ai : struct_AI;
  END_VAR
  VAR_IN_OUT
    on1Temperature : struct_AnalogParametr;
    on2Temperature : struct_AnalogParametr;
    hystereses : struct_AnalogParametr;
  END_VAR
  VAR
    _sunpackerCommand : fb_sunpackerCommand;
    _statusAi : TYPE_StatusAi;
    _statusDualInput : TYPE_statusDualInput;
    _commandDualInput : TYPE_commandDualInput;
    source : BYTE;
    cmd : BYTE;
    lastCmd : BYTE;
    source_for_Status : BYTE;
    cmd_for_Status : BYTE;
    command_error_for_Status : BYTE;
    resetCmdTimer : TON;
    resetCmdTimerPriznak : BOOL;
    onInit : BOOL;
  END_VAR

  IF NOT onInit THEN
  StrAlg.inCanRun:=TRUE;
  onInit:=TRUE;
  END_IF;

  IF StrAlg.isRuning THEN

  StrAlg.hasError := im1.CommandFault OR im2.CommandFault OR (ai.interval<_statusAi.normal);

      IF (ai.interval>=_statusAi.normal) THEN

            IF (ai.value>= on1Temperature.Value) THEN
                IF im1.onStatus <> _statusDualInput.STATUS_ON THEN
  	       im1.inCommand_Alg:=BYTE_TO_WORD(_commandDualInput.CMD_ON); (*cmd_on*)
                END_IF;
            END_IF;

            IF  ai.value < (on1Temperature.Value - hystereses.Value) THEN
                IF im1.onStatus <> _statusDualInput.STATUS_OFF THEN
  	       im1.inCommand_Alg:=BYTE_TO_WORD(_commandDualInput.CMD_OFF);
                END_IF;
            END_IF;

             IF (ai.value>= on2Temperature.Value) THEN
                IF im2.onStatus <> _statusDualInput.STATUS_ON THEN
  	       im2.inCommand_Alg:=BYTE_TO_WORD(_commandDualInput.CMD_ON); (*cmd_on*)
                END_IF;
            END_IF;

            IF  ai.value < (on2Temperature.Value - hystereses.Value) THEN
                IF im2.onStatus <> _statusDualInput.STATUS_OFF THEN
  	       im2.inCommand_Alg:=BYTE_TO_WORD(_commandDualInput.CMD_OFF);
                END_IF;
            END_IF;
       END_IF;

  END_IF;

  StrAlg.CanRun := StrAlg.inCanRun;

  StrAlg.OpcCommandsDisabled := StrAlg.inOpcCommandsDisabled;

  (* ---- Если управление с ВУ заблокировано, то  передаем команду из алгоритма ---- *)
  IF StrAlg.inOpcCommandsDisabled THEN
  	StrAlg.inCommand := StrAlg.inCommand_Alg;
  ELSE (* иначе передаем команду с АРМа*)
  	StrAlg.inCommand := StrAlg.inCommand_ARM;
  END_IF;

  _sunpackerCommand(command := StrAlg.inCommand);
  	source := _sunpackerCommand.source;
  	cmd := _sunpackerCommand.cmd;

  IF cmd <> 0 AND lastCmd <> cmd AND (((NOT StrAlg.opcCommandsDisabled) AND source > 0) OR source = 0) then
  	CASE BYTE_TO_INT(cmd) OF
  		(*cmdRun*) 1: 	IF (StrAlg.CanRun) THEN
  					StrAlg.isRuning := TRUE;
  					StrAlg.isEnded := FALSE;
  					StrAlg.hasError := FALSE;
                                                    StrAlg.opcCommandsDisabled:=FALSE;
  					im1.inOpcCommandsDisabled:=TRUE;
                                                    im2.inOpcCommandsDisabled:=TRUE;
  					cmd_for_Status := cmd;
  					source_for_Status := source;
  					command_error_for_Status := 0;
  				ELSE
  					StrAlg.isRuning := FALSE;
  					StrAlg.isEnded := FALSE;
  					StrAlg.hasError 	:= FALSE;

  					cmd_for_Status := 0;
  					source_for_Status := source;
  					command_error_for_Status := cmd;
  				END_IF;
  		(*cmdReset*) 2: 	StrAlg.isRuning := FALSE;
  				StrAlg.isEnded := FALSE;
  				StrAlg.hasError 	:= FALSE;
                                          StrAlg.opcCommandsDisabled:=FALSE;
                                          im1.inOpcCommandsDisabled:=FALSE;
                                          im2.inOpcCommandsDisabled:=FALSE;
                                          im1.inCommand_Alg:=0;
                                          im2.inCommand_Alg:=0;
  				cmd_for_Status := cmd;
  				source_for_Status := source;
  				command_error_for_Status := 0;
  	END_CASE;
  	resetCmdTimer(IN := false);
  	resetCmdTimerPriznak := TRUE;
  END_IF;
  lastCmd := cmd;

  resetCmdTimer(IN := resetCmdTimerPriznak, PT := T#5S);
  IF resetCmdTimer.Q THEN
  	resetCmdTimerPriznak := FALSE;
  	source_for_Status := 0;
  	cmd_for_Status := 0;
  	command_error_for_Status := 0;
  END_IF;

  (*TODO: TYPE PROGRAM CODE HERE*)
  StrAlg.status :=  SHL(BYTE_TO_DWORD(source_for_Status), 29)
  			OR SHL(BYTE_TO_DWORD(cmd_for_Status), 26)
  			OR SHL(BYTE_TO_DWORD(command_error_for_Status), 23)
  			OR SHL(BOOL_TO_DWORD(StrAlg.OpcCommandsDisabled ), 21)
  			OR SHL(BOOL_TO_DWORD(StrAlg.hasError),4)
  			OR SHL(BOOL_TO_DWORD(StrAlg.CanRun),2)
  			OR SHL(BOOL_TO_DWORD(StrAlg.isEnded),1)
  			OR BOOL_TO_DWORD(StrAlg.isRuning);
END_FUNCTION_BLOCK

FUNCTION_BLOCK fb_AutoNUAlg
  VAR_IN_OUT
    StrAlg : struct_Alg;
    nu1 : struct_OilPump;
    nu2 : struct_OilPump;
  END_VAR
  VAR_INPUT
    dPoil : struct_AI;
  END_VAR
  VAR_IN_OUT
    mainNU : struct_DiscretParametr;
  END_VAR
  VAR_EXTERNAL
    Reset_HasNU : BOOL;
  END_VAR
  VAR_IN_OUT
    Lowdp_di : struct_singleSignal;
    Ust_Swap : struct_AnalogParametr;
  END_VAR
  VAR
    _prevMainNU : UINT;
    _sunpackerCommand : fb_sunpackerCommand;
    _statusAi : TYPE_StatusAi;
    _statusDualInput : TYPE_statusDualInput;
    _commandDualInput : TYPE_commandDualInput;
    source : BYTE;
    cmd : BYTE;
    lastCmd : BYTE;
    source_for_Status : BYTE;
    cmd_for_Status : BYTE;
    command_error_for_Status : BYTE;
    resetCmdTimer : TON;
    waitPressure : TON;
    waitPressureTrig : R_TRIG;
    resetCmdTimerPriznak : BOOL;
    onInit : BOOL;
    onStart : BOOL;
  END_VAR
  VAR_EXTERNAL
    NotHasRezervNU : BOOL;
  END_VAR

  IF NOT onInit THEN
  StrAlg.inCanRun:=TRUE;
  StrAlg.inOpcCommandsDisabled:=TRUE;
  (*nu1.Osnovnoy:=TRUE; nu2.Osnovnoy:=FALSE;*)
  onInit:=TRUE;
  END_IF;

  IF Reset_HasNU THEN
  nu1.inBlocked:=FALSE;
  nu2.inBlocked:=FALSE;
  END_IF;

  NotHasRezervNU:=(nu1.Blocked OR nu2.Blocked);

  IF StrAlg.isRuning THEN

  StrAlg.hasError := nu1.CommandFault OR nu2.CommandFault OR (dPoil.interval<_statusAi.normal);

   IF mainNU.value<>_prevMainNU OR NOT onStart THEN

          CASE mainNU.value OF
  	0: nu1.Osnovnoy:=TRUE; nu2.Osnovnoy:=FALSE;
  	1: nu1.Osnovnoy:=FALSE; nu2.Osnovnoy:=TRUE;

          END_CASE;

      IF  nu1.Osnovnoy AND NOT nu1.Blocked THEN
          nu1.inCommand_Alg:=BYTE_TO_WORD(_commandDualInput.CMD_ON);
      ELSIF NOT NotHasRezervNU THEN
          nu1.inCommand_Alg:=BYTE_TO_WORD(_commandDualInput.CMD_OFF);
      END_IF;

      IF  nu2.Osnovnoy AND NOT nu2.Blocked THEN
          nu2.inCommand_Alg:=BYTE_TO_WORD(_commandDualInput.CMD_ON);
       ELSIF NOT NotHasRezervNU THEN
          nu2.inCommand_Alg:=BYTE_TO_WORD(_commandDualInput.CMD_OFF);
      END_IF;
        onStart:=TRUE;
       _prevMainNU:=mainNU.value;
   END_IF;

    (*IF (nu1.onStatus = _statusDualInput.STATUS_On) OR (nu2.onStatus = _statusDualInput.STATUS_On) THEN*)
      (*Если через 5С насос не нагнал 100кПа масла - он сломался и надо переключить насос*)
      IF dPoil.interval>= _statusAi.NORMAL THEN
            waitPressure(IN:=(dPoil.value<Ust_Swap.Value OR LowdP_DI.q) AND NOT NotHasRezervNU, PT:= T#5S);
      ELSE
  	waitPressure(IN:=(FALSE));
      END_IF;

      waitPressureTrig(CLK:=waitPressure.Q);
      IF waitPressureTrig.Q THEN
  	(*IF nu1.onStatus = _statusDualInput.STATUS_ON THEN*)
             IF mainNU.value = 0 THEN
  		nu1.inBlocked:=TRUE;
                      nu1.inCommand_Alg:=BYTE_TO_WORD(_commandDualInput.CMD_OFF);
  			(*IF 	mainNU.value = 0 THEN*)
                                          setValue(mainNU, 1);
  			(*END_IF;*)
  	END_IF;

  	(*IF nu2.onStatus = _statusDualInput.STATUS_ON THEN*)
            IF mainNU.value = 1 THEN
  		nu2.inBlocked:=TRUE;
                      nu2.inCommand_Alg:=BYTE_TO_WORD(_commandDualInput.CMD_OFF);
  			(*IF 	mainNU.value = 1 THEN*)
  				setValue(mainNU, 0);
  			(*END_IF;*)
  	END_IF;
      END_IF;
   (* END_IF;*)

  END_IF;

  StrAlg.CanRun := StrAlg.inCanRun;

  StrAlg.OpcCommandsDisabled := StrAlg.inOpcCommandsDisabled;

  (* ---- Если управление с ВУ заблокировано, то  передаем команду из алгоритма ---- *)
  IF StrAlg.inOpcCommandsDisabled THEN
  	StrAlg.inCommand := StrAlg.inCommand_Alg;
  ELSE (* иначе передаем команду с АРМа*)
  	StrAlg.inCommand := StrAlg.inCommand_ARM;
  END_IF;

  _sunpackerCommand(command := StrAlg.inCommand);
  	source := _sunpackerCommand.source;
  	cmd := _sunpackerCommand.cmd;

  IF cmd <> 0 AND lastCmd <> cmd AND (((NOT StrAlg.opcCommandsDisabled) AND source > 0) OR source = 0) then
  	CASE BYTE_TO_INT(cmd) OF
  		(*cmdRun*) 1: 	IF (StrAlg.CanRun) THEN
  					StrAlg.isRuning := TRUE;
  					StrAlg.isEnded := FALSE;
  					StrAlg.hasError := FALSE;

                                                    (*****************       OnRun       *****************)
  					nu1.inOpcCommandsDisabled:=TRUE;
                                                    nu2.inOpcCommandsDisabled:=TRUE;

  					cmd_for_Status := cmd;
  					source_for_Status := source;
  					command_error_for_Status := 0;
  				ELSE
  					StrAlg.isRuning := FALSE;
  					StrAlg.isEnded := FALSE;
  					StrAlg.hasError 	:= FALSE;

  					cmd_for_Status := 0;
  					source_for_Status := source;
  					command_error_for_Status := cmd;
  				END_IF;
  		(*cmdReset*) 2: 	StrAlg.isRuning := FALSE;
  				StrAlg.isEnded := FALSE;
  				StrAlg.hasError 	:= FALSE;

                                          (*****************       OnReset       *****************)
                                          waitPressure(IN:=(FALSE));
                                          onStart:=FALSE;

  				cmd_for_Status := cmd;
  				source_for_Status := source;
  				command_error_for_Status := 0;
  	END_CASE;
  	resetCmdTimer(IN := false);
  	resetCmdTimerPriznak := TRUE;
  END_IF;
  lastCmd := cmd;

  resetCmdTimer(IN := resetCmdTimerPriznak, PT := T#5S);
  IF resetCmdTimer.Q THEN
  	resetCmdTimerPriznak := FALSE;
  	source_for_Status := 0;
  	cmd_for_Status := 0;
  	command_error_for_Status := 0;
  END_IF;

  (*TODO: TYPE PROGRAM CODE HERE*)
  StrAlg.status :=  SHL(BYTE_TO_DWORD(source_for_Status), 29)
  			OR SHL(BYTE_TO_DWORD(cmd_for_Status), 26)
  			OR SHL(BYTE_TO_DWORD(command_error_for_Status), 23)
  			OR SHL(BOOL_TO_DWORD(StrAlg.OpcCommandsDisabled ), 21)
                                OR SHL(BOOL_TO_DWORD(NotHasRezervNU), 15)
  			OR SHL(BOOL_TO_DWORD(StrAlg.hasError),4)
  			OR SHL(BOOL_TO_DWORD(StrAlg.CanRun),2)
  			OR SHL(BOOL_TO_DWORD(StrAlg.isEnded),1)
  			OR BOOL_TO_DWORD(StrAlg.isRuning);
END_FUNCTION_BLOCK

FUNCTION_BLOCK fb_AutoPnsAlg
  VAR_IN_OUT
    StrAlg : struct_Alg;
    Nasos : struct_Switch;
  END_VAR
  VAR_INPUT
    diPlow : struct_singleSignal;
    Poil : struct_AI;
    Ust_Run : struct_AnalogParametr;
    Ust_Stop : struct_AnalogParametr;
  END_VAR
  VAR
    _sunpackerCommand : fb_sunpackerCommand;
    _statusAi : TYPE_StatusAi;
    _statusDualInput : TYPE_statusDualInput;
    _commandDualInput : TYPE_commandDualInput;
    source : BYTE;
    cmd : BYTE;
    lastCmd : BYTE;
    source_for_Status : BYTE;
    cmd_for_Status : BYTE;
    command_error_for_Status : BYTE;
    resetCmdTimer : TON;
    resetCmdTimerPriznak : BOOL;
    onInit : BOOL;
    onTrig : R_TRIG;
    offTrig : R_TRIG;
    waitOn : TON;
    waitOff : TON;
  END_VAR
  VAR_EXTERNAL
    AlgTimers : struct_AlgTimers;
  END_VAR

  IF NOT onInit THEN
  StrAlg.inOpcCommandsDisabled:=TRUE;
  StrAlg.inCanRun:=TRUE;
  onInit:=TRUE;
  END_IF;

  IF StrAlg.isRuning THEN

  StrAlg.hasError := Nasos.CommandFault OR (Poil.interval < _statusAi.normal OR NOT diPlow.reliability);

      IF (Poil.Interval >= _statusAi.normal) THEN
      waitOn(IN:=Poil.Value <= Ust_Run.value OR diPlow.q, PT := T#1S);
      waitOff(IN:= Poil.Value >= Ust_Stop.value, PT := T#300S);

      ELSE
      waitOn(IN:=diPlow.Q, PT := T#1S);
      END_IF;

  onTrig(CLK:=waitOn.Q);
  offTrig(CLK:=waitOff.Q);

      IF onTrig.Q THEN
      Nasos.inopcCommandsDisabled:=TRUE;
      Nasos.inCommand_Alg:=BYTE_TO_WORD(_commandDualInput.CMD_ON);
      END_IF;

      IF offTrig.Q THEN
          IF NOT (Nasos.onStatus=_statusDualInput.STATUS_OFF) THEN
          Nasos.inopcCommandsDisabled:=TRUE;
          Nasos.inCommand_Alg:=BYTE_TO_WORD(_commandDualInput.CMD_OFF);
          END_IF;
      END_IF;

      IF (Poil.Value>=Ust_Stop.value) AND Nasos.inopcCommandsDisabled AND (Nasos.onStatus=_statusDualInput.STATUS_OFF) THEN
          Nasos.inopcCommandsDisabled:=FALSE;
      END_IF;

  AlgTimers.AutoPns_OnTimer:=UDINT_TO_UINT(TIME_TO_UDINT(waitOn.PT - waitOn.ET)/1000);
  AlgTimers.AutoPns_OffTimer:=UDINT_TO_UINT(TIME_TO_UDINT(waitOff.PT -waitOff.ET)/1000);

  END_IF;

  StrAlg.CanRun := StrAlg.inCanRun;

  StrAlg.OpcCommandsDisabled := StrAlg.inOpcCommandsDisabled;

  (* ---- Если управление с ВУ заблокировано, то  передаем команду из алгоритма ---- *)
  IF StrAlg.inOpcCommandsDisabled THEN
  	StrAlg.inCommand := StrAlg.inCommand_Alg;
  ELSE (* иначе передаем команду с АРМа*)
  	StrAlg.inCommand := StrAlg.inCommand_ARM;
  END_IF;

  _sunpackerCommand(command := StrAlg.inCommand);
  	source := _sunpackerCommand.source;
  	cmd := _sunpackerCommand.cmd;

  IF cmd <> 0 AND lastCmd <> cmd AND (((NOT StrAlg.opcCommandsDisabled) AND source > 0) OR source = 0) then
  	CASE BYTE_TO_INT(cmd) OF
  		(*cmdRun*) 1: 	IF (StrAlg.CanRun) THEN
  					StrAlg.isRuning := TRUE;
  					StrAlg.isEnded := FALSE;
  					StrAlg.hasError := FALSE;
  					(*****************       OnRun       *****************)

  					cmd_for_Status := cmd;
  					source_for_Status := source;
  					command_error_for_Status := 0;
  				ELSE
  					StrAlg.isRuning := FALSE;
  					StrAlg.isEnded := FALSE;
  					StrAlg.hasError 	:= FALSE;

  					cmd_for_Status := 0;
  					source_for_Status := source;
  					command_error_for_Status := cmd;
  				END_IF;
  		(*cmdReset*) 2: 	StrAlg.isRuning := FALSE;
  				StrAlg.isEnded := FALSE;
  				StrAlg.hasError 	:= FALSE;

                                           (*****************       OnReset       *****************)
                                          waitOn(in:=FALSE);
                                          waitOff(in:=FALSE);
                                          AlgTimers.AutoPns_OffTimer:=UDINT_TO_UINT(TIME_TO_UDINT(waitOff.pt -waitOff.ET)/1000);

  				cmd_for_Status := cmd;
  				source_for_Status := source;
  				command_error_for_Status := 0;
  	END_CASE;
  	resetCmdTimer(IN := false);
  	resetCmdTimerPriznak := TRUE;
  END_IF;
  lastCmd := cmd;

  resetCmdTimer(IN := resetCmdTimerPriznak, PT := T#5S);
  IF resetCmdTimer.Q THEN
  	resetCmdTimerPriznak := FALSE;
  	source_for_Status := 0;
  	cmd_for_Status := 0;
  	command_error_for_Status := 0;
  END_IF;

  (*TODO: TYPE PROGRAM CODE HERE*)
  StrAlg.status :=  SHL(BYTE_TO_DWORD(source_for_Status), 29)
  			OR SHL(BYTE_TO_DWORD(cmd_for_Status), 26)
  			OR SHL(BYTE_TO_DWORD(command_error_for_Status), 23)
  			OR SHL(BOOL_TO_DWORD(StrAlg.OpcCommandsDisabled ), 21)
  			OR SHL(BOOL_TO_DWORD(StrAlg.hasError),4)
  			OR SHL(BOOL_TO_DWORD(StrAlg.CanRun),2)
  			OR SHL(BOOL_TO_DWORD(StrAlg.isEnded),1)
  			OR BOOL_TO_DWORD(StrAlg.isRuning);
END_FUNCTION_BLOCK

FUNCTION_BLOCK fb_AutoTenAlg
  VAR_IN_OUT
    StrAlg : struct_Alg;
    PNS : struct_Switch;
    TEN : struct_Switch;
  END_VAR
  VAR_INPUT
    T_masla : struct_AI;
    Uroven_masla : struct_AI;
    offTemperature : struct_AnalogParametr;
  END_VAR
  VAR
    _sunpackerCommand : fb_sunpackerCommand;
    _statusAi : TYPE_StatusAi;
    _statusDualInput : TYPE_statusDualInput;
    _commandDualInput : TYPE_commandDualInput;
    source : BYTE;
    cmd : BYTE;
    lastCmd : BYTE;
    source_for_Status : BYTE;
    cmd_for_Status : BYTE;
    command_error_for_Status : BYTE;
    resetCmdTimer : TON;
    resetCmdTimerPriznak : BOOL;
    onInit : BOOL;
  END_VAR

  IF NOT onInit THEN
  StrAlg.inCanRun:=TRUE;
  onInit:=TRUE;
  END_IF;

  IF StrAlg.isRuning THEN

  IF ((T_masla.interval >= _statusAi.normal) AND (T_masla.value > offTemperature.Value)) OR
  ((Uroven_masla.interval >= _statusAi.normal) AND (Uroven_masla.value < Uroven_masla.LA)) OR
  (PNS.onStatus=_statusDualInput.STATUS_OFF) THEN

        TEN.inOpcCommandsDisabled:=TRUE;

  	IF TEN.onStatus = _statusDualInput.STATUS_ON THEN
            TEN.inCommand_Alg:=BYTE_TO_WORD(_commandDualInput.CMD_OFF);
  	END_IF;

  ELSIF PNS.onStatus = _statusDualInput.STATUS_ON THEN
        TEN.inOpcCommandsDisabled:=FALSE;
  END_IF;

  END_IF;

  StrAlg.CanRun := StrAlg.inCanRun;
  StrAlg.hasError := TEN.CommandFault OR (T_masla.interval < _statusAi.normal) OR (Uroven_masla.interval < _statusAi.normal);

  StrAlg.OpcCommandsDisabled := StrAlg.inOpcCommandsDisabled;

  (* ---- Если управление с ВУ заблокировано, то  передаем команду из алгоритма ---- *)
  IF StrAlg.inOpcCommandsDisabled THEN
  	StrAlg.inCommand := StrAlg.inCommand_Alg;
  ELSE (* иначе передаем команду с АРМа*)
  	StrAlg.inCommand := StrAlg.inCommand_ARM;
  END_IF;

  _sunpackerCommand(command := StrAlg.inCommand);
  	source := _sunpackerCommand.source;
  	cmd := _sunpackerCommand.cmd;

  IF cmd <> 0 AND lastCmd <> cmd AND (((NOT StrAlg.opcCommandsDisabled) AND source > 0) OR source = 0) then
  	CASE BYTE_TO_INT(cmd) OF
  		(*cmdRun*) 1: 	IF StrAlg.CanRun AND NOT StrAlg.hasError THEN
  					StrAlg.isRuning := TRUE;
  					StrAlg.isEnded := FALSE;
  					(*StrAlg.hasError := FALSE;*)

                                                    (*****************       OnRun       *****************)
                                                    IF StrAlg.inOpcCommandsDisabled THEN
  		                              StrAlg.inOpcCommandsDisabled:=FALSE;
                                                    END_IF;
  					cmd_for_Status := cmd;
  					source_for_Status := source;
  					command_error_for_Status := 0;
  				ELSE
  					StrAlg.isRuning := FALSE;
  					StrAlg.isEnded := FALSE;
  					(*StrAlg.hasError 	:= FALSE;*)

  					cmd_for_Status := 0;
  					source_for_Status := source;
  					command_error_for_Status := cmd;
  				END_IF;
  		(*cmdReset*) 2: 	StrAlg.isRuning := FALSE;
  				StrAlg.isEnded := FALSE;
  				(*StrAlg.hasError 	:= FALSE;*)

                                          (*****************       OnReset       *****************)
                                          TEN.inOpcCommandsDisabled:=TRUE;
                                          TEN.inCommand_Alg:=BYTE_TO_WORD(_commandDualInput.CMD_OFF);

  				cmd_for_Status := cmd;
  				source_for_Status := source;
  				command_error_for_Status := 0;
  	END_CASE;
  	resetCmdTimer(IN := false);
  	resetCmdTimerPriznak := TRUE;
  END_IF;
  lastCmd := cmd;

  resetCmdTimer(IN := resetCmdTimerPriznak, PT := T#5S);
  IF resetCmdTimer.Q THEN
  	resetCmdTimerPriznak := FALSE;
  	source_for_Status := 0;
  	cmd_for_Status := 0;
  	command_error_for_Status := 0;
  END_IF;

  (*TODO: TYPE PROGRAM CODE HERE*)
  StrAlg.status :=  SHL(BYTE_TO_DWORD(source_for_Status), 29)
  			OR SHL(BYTE_TO_DWORD(cmd_for_Status), 26)
  			OR SHL(BYTE_TO_DWORD(command_error_for_Status), 23)
  			OR SHL(BOOL_TO_DWORD(StrAlg.OpcCommandsDisabled ), 21)
  			OR SHL(BOOL_TO_DWORD(StrAlg.hasError),4)
  			OR SHL(BOOL_TO_DWORD(StrAlg.CanRun),2)
  			OR SHL(BOOL_TO_DWORD(StrAlg.isEnded),1)
  			OR BOOL_TO_DWORD(StrAlg.isRuning);
END_FUNCTION_BLOCK

FUNCTION_BLOCK fb_BaseAlgoritm
  VAR_IN_OUT
    StrAlg : struct_Alg;
  END_VAR
  VAR
    _sunpackerCommand : fb_sunpackerCommand;
    source : BYTE;
    cmd : BYTE;
    lastCmd : BYTE;
    source_for_Status : BYTE;
    cmd_for_Status : BYTE;
    command_error_for_Status : BYTE;
    resetCmdTimer : TON;
    resetCmdTimerPriznak : BOOL;
  END_VAR

  StrAlg.CanRun := StrAlg.inCanRun;
  StrAlg.hasError := StrAlg.inHasError OR (command_error_for_Status <> 0);
  StrAlg.isEnded := StrAlg.inEnded;

  StrAlg.OpcCommandsDisabled := StrAlg.inOpcCommandsDisabled;

  (* ---- Если управление с ВУ заблокировано, то передаем команду из алгоритма ---- *)
  IF StrAlg.inOpcCommandsDisabled THEN
  	StrAlg.inCommand := StrAlg.inCommand_Alg;
  ELSE (* иначе передаем команду с АРМа*)
  	StrAlg.inCommand := StrAlg.inCommand_ARM;
  END_IF;

  _sunpackerCommand(command := StrAlg.inCommand);
  	source := _sunpackerCommand.source;
  	cmd := _sunpackerCommand.cmd;

  IF cmd <> 0 AND lastCmd <> cmd AND (((NOT StrAlg.opcCommandsDisabled) AND source > 0) OR source = 0) then
  	CASE BYTE_TO_INT(cmd) OF
  		(*cmdRun*) 1: 	IF (StrAlg.CanRun) THEN
  					StrAlg.isRuning := TRUE;
  					StrAlg.isEnded := FALSE;
  					StrAlg.hasError 	:= FALSE;

  					cmd_for_Status := cmd;
  					source_for_Status := source;
  					command_error_for_Status := 0;
  				ELSE
  					StrAlg.isRuning := FALSE;
  					StrAlg.isEnded := FALSE;
  					StrAlg.hasError 	:= FALSE;

  					cmd_for_Status := 0;
  					source_for_Status := source;
  					command_error_for_Status := cmd;
  				END_IF;
  		(*cmdReset*) 2: 	StrAlg.isRuning := FALSE;
  				StrAlg.isEnded := FALSE;
  				StrAlg.hasError 	:= FALSE;
  				cmd_for_Status := cmd;
  				source_for_Status := source;
  				command_error_for_Status := 0;
  	END_CASE;
  	resetCmdTimer(IN := false);
  	resetCmdTimerPriznak := TRUE;
  END_IF;
  lastCmd := cmd;

  resetCmdTimer(IN := resetCmdTimerPriznak, PT := T#5S);
  IF resetCmdTimer.Q THEN
  	resetCmdTimerPriznak := FALSE;
  	source_for_Status := 0;
  	cmd_for_Status := 0;
  	command_error_for_Status := 0;
  END_IF;

  StrAlg.status :=  SHL(BYTE_TO_DWORD(source_for_Status), 29)
  			OR SHL(BYTE_TO_DWORD(cmd_for_Status), 26)
  			OR SHL(BYTE_TO_DWORD(command_error_for_Status), 23)
  			OR SHL(BOOL_TO_DWORD(StrAlg.OpcCommandsDisabled ), 21)
  			OR SHL(BOOL_TO_DWORD(StrAlg.hasError),4)
  			OR SHL(BOOL_TO_DWORD(StrAlg.CanRun),2)
  			OR SHL(BOOL_TO_DWORD(StrAlg.isEnded),1)
  			OR BOOL_TO_DWORD(StrAlg.isRuning);
END_FUNCTION_BLOCK

FUNCTION_BLOCK fb_BaseProtection
  VAR
    inSignaling : BOOL;
    inTag : BYTE;
    inRunOnStart : BOOL;
    inCanRun : BOOL;
    inHasError : BOOL;
    inEnded : BOOL;
    inOpcCommandsDisabled : BOOL;
    inCommand : WORD;
    Tag : BYTE;
    status : DWORD;
    CanRun : BOOL;
    OpcCommandsDisabled : BOOL;
    isRunning : BOOL;
    HasError : BOOL;
    isEnded : BOOL;
    Remont : BOOL;
    Check : BOOL;
    Signaling : BOOL;
    SignalingTP : BOOL;
    RunOnStart : BOOL;
    _sunpackerCommand : fb_sunpackerCommand;
    _ProtectionTags : TYPE_ProtectionTags;
    _signalingTp : TOF;
    source : BYTE;
    cmd : BYTE;
    lastCmd : BYTE;
    source_for_Status : BYTE;
    cmd_for_Status : BYTE;
    command_error_for_Status : BYTE;
    resetCmdTimer : TON;
    resetCmdTimerPriznak : BOOL;
    signalinTimer : TON;
    runOnStart_Trig : R_TRIG;
  END_VAR

  Tag := inTag;
  RunOnStart := inRunOnStart;

  CanRun := inCanRun;
  hasError := inHasError;
  isEnded := inEnded;

  OpcCommandsDisabled := inOpcCommandsDisabled;

  _sunpackerCommand(command := inCommand);
  	source := _sunpackerCommand.source;
  	cmd := _sunpackerCommand.cmd;

  IF cmd <> 0 AND lastCmd <> cmd AND (((NOT opcCommandsDisabled) AND source > 0) OR source = 0) then
  	CASE BYTE_TO_INT(cmd) OF
  		(*cmdRun*) 1: 	IF CanRun AND NOT Remont THEN
  					isEnded := FALSE;
  					hasError 	:= FALSE;
  					isRunning := TRUE;
  					cmd_for_Status := cmd;
  					source_for_Status := source;
  					command_error_for_Status := 0;
  				ELSE
  					isRunning := FALSE;
  					isEnded := FALSE;
  					hasError 	:= FALSE;

  					cmd_for_Status := 0;
  					source_for_Status := source;
  					command_error_for_Status := cmd;
  				END_IF;
  		(*cmdReset*) 2: 	isRunning := FALSE;
  				isEnded := FALSE;
  				hasError 	:= FALSE;
  				inSignaling := FALSE;
  				Check := FALSE;
  				cmd_for_Status := cmd;
  				source_for_Status := source;
  				command_error_for_Status := 0;
  	(*cmd_setRemont*) 4 :	Remont := TRUE;
  				isRunning := FALSE;

  				cmd_for_Status := cmd;
  				source_for_Status := source;
  				command_error_for_Status := 0;
  	(*cmd_resetRemont*) 5 : 	IF inSignaling THEN
  					cmd_for_Status := 0;
  					source_for_Status := 0;
  					command_error_for_Status := cmd;
  				ELSE
  					Remont := FALSE;
  					isRunning := TRUE;

  					cmd_for_Status := cmd;
  					source_for_Status := source;
  					command_error_for_Status := 0;
  				END_IF;
  	(*cmd_setCheck*) 6 : 	Check := TRUE;

  				cmd_for_Status := cmd;
  				source_for_Status := source;
  				command_error_for_Status := 0;
  	END_CASE;
  	resetCmdTimer(IN := false);
  	resetCmdTimerPriznak := TRUE;
  END_IF;
  lastCmd := cmd;

  resetCmdTimer(IN := resetCmdTimerPriznak);
  IF resetCmdTimer.Q THEN
  	resetCmdTimerPriznak := FALSE;
  	source_for_Status := 0;
  	cmd_for_Status := 0;
  	command_error_for_Status := 0;
  END_IF;

  IF isRunning THEN
  	Signaling := inSignaling;
  	SignalingTP := _signalingTp.Q;
  ELSE
  	Signaling := 0;
  	SignalingTP := 0;
  END_IF;

  IF NOT Remont AND NOT Check THEN
  	_signalingTp(in := Signaling, PT := T#1s);
  ELSE
  	_signalingTp(in := FALSE);
  END_IF;

  status :=  SHL(BYTE_TO_DWORD(source_for_Status), 29)
  			OR SHL(BYTE_TO_DWORD(cmd_for_Status), 26)
  			OR SHL(BYTE_TO_DWORD(command_error_for_Status), 23)
  			OR SHL(BOOL_TO_DWORD(OpcCommandsDisabled ), 21)
  			OR SHL(BOOL_TO_DWORD(Signaling), 16)
  			OR SHL(BOOL_TO_DWORD(RunOnStart ), 15)
  			OR SHL(BOOL_TO_DWORD(remont), 6)
  			OR SHL(BOOL_TO_DWORD(Check), 5)
  			OR SHL(BOOL_TO_DWORD(hasError), 4)
  			OR SHL(BOOL_TO_DWORD(SignalingTP), 3)
  			OR SHL(BOOL_TO_DWORD(CanRun), 2)
  			OR SHL(BOOL_TO_DWORD(isEnded), 1)
  			OR BOOL_TO_DWORD(isRunning);
END_FUNCTION_BLOCK

FUNCTION_BLOCK fb_DI_Init
  VAR_INPUT
    data_Ini : BOOL;
    imit : BOOL         := FALSE;
  END_VAR
  VAR_IN_OUT
    strDI : struct_DI;
  END_VAR
  VAR_OUTPUT
    Init : BOOL         := FALSE;
  END_VAR

  (*****            Функциональный блок переинициализации структуры-дескриптора канала дискретного ввода        *****)

   Init := FALSE;

      IF data_Ini THEN                            (* Параметрам требуется переинициализация. *)
          strDI.imit       := imit;
          data_Ini:=FALSE;
          Init := TRUE;
      END_IF;
    IF Init THEN
  imit:=FALSE;
      END_IF;
END_FUNCTION_BLOCK

FUNCTION_BLOCK fb_DOSourceMlp
  VAR_IN_OUT
    arDout : TWordData;
  END_VAR
  VAR_INPUT
    err_mod : TItemDIN;
  END_VAR
  VAR_IN_OUT
    strDO : struct_DO;
  END_VAR
  VAR
    bitNumber : INT;
  END_VAR

  strDO.blConnect := TRUE; (*((UINT_TO_WORD(err_mod.wValue) = 20) and (UINT_TO_WORD(err_mod.wFlags) = 192));*)

  strDO.value:=0;

  FOR bitNumber:=0 TO 15 BY 1 DO
  	strDO.value:=strDO.value OR (SHL(BOOL_TO_WORD(strDO.bits[bitNumber]),bitNumber));
  END_FOR;

  IF NOT strDO.imit THEN
  	 arDout.wValue:= WORD_TO_UINT(strDO.value);
  END_IF;
END_FUNCTION_BLOCK

FUNCTION_BLOCK fb_DO_Init
  VAR_INPUT
    data_Ini : BOOL;
    imit : BOOL         := FALSE;
  END_VAR
  VAR_IN_OUT
    strDO : struct_DO;
  END_VAR
  VAR_OUTPUT
    Init : BOOL         := FALSE;
  END_VAR

  (*****            Функциональный блок переинициализации структуры-дескриптора канала дискретного ввода.            *****)
   Init := FALSE;

      IF data_Ini THEN                            (* Параметрам требуется переинициализация. *)
          strDO.imit       := imit;
          data_Ini:=FALSE;
          Init := TRUE;
      END_IF;
    IF Init THEN
  imit:=FALSE;
     END_IF;
END_FUNCTION_BLOCK

FUNCTION_BLOCK fb_DiProtection
  VAR_INPUT
    di : struct_singleSignal;
  END_VAR
  VAR_IN_OUT
    StrDIp : struct_DiProtection;
  END_VAR
  VAR
    _sunpackerCommand : fb_sunpackerCommand;
    _ProtectionTags : TYPE_ProtectionTags;
    _signalingTp : TOF;
    timer : TON;
    SignalingTrig : R_TRIG;
    SignalingFTrig : F_TRIG;
    SignalingDi : BOOL;
    source : BYTE;
    cmd : BYTE;
    lastCmd : BYTE;
    source_for_Status : BYTE;
    cmd_for_Status : BYTE;
    command_error_for_Status : BYTE;
    resetCmdTimer : TON;
    resetCmdTimerPriznak : BOOL;
    signalinTimer : TON;
    runOnStart_Trig : R_TRIG;
  END_VAR

  timer(IN := di.Q AND StrDIp.isRunning  , PT := StrDIp.delay);
  SignalingTrig(CLK := timer.Q);
  IF SignalingTrig.Q THEN
  	SignalingDi := TRUE;
  END_IF;
  SignalingFTrig(CLK := timer.Q);
  IF SignalingFTrig.Q THEN
  	SignalingDi := FALSE;
  END_IF;

  StrDIp.Tag := StrDIp.inTag;
  StrDIp.RunOnStart := StrDIp.inRunOnStart;

  StrDIp.CanRun := StrDIp.inCanRun;

  StrDIp.OpcCommandsDisabled := StrDIp.inOpcCommandsDisabled;

  (* ---- Если управление с ВУ заблокировано, то передаем команду из алгоритма ---- *)
  IF StrDIp.inOpcCommandsDisabled THEN
  	StrDIp.inCommand := StrDIp.inCommand_Alg;
  ELSE (* иначе передаем команду с АРМа*)
  	StrDIp.inCommand := StrDIp.inCommand_ARM;
  END_IF;

  _sunpackerCommand(command := StrDIp.inCommand);
  	source := _sunpackerCommand.source;
  	cmd := _sunpackerCommand.cmd;

  IF cmd <> 0 AND lastCmd <> cmd AND (((NOT StrDIp.opcCommandsDisabled) AND source > 0) OR source = 0) then

  	CASE BYTE_TO_INT(cmd) OF
  	        (*cmdRun*) 1: 	IF        NOT StrDIp.Remont THEN
  					StrDIp.isEnded := FALSE;
  					StrDIp.hasError 	:= FALSE;
  					StrDIp.isRunning := TRUE;
  					cmd_for_Status := cmd;
  					source_for_Status := source;
  					command_error_for_Status := 0;
  				ELSE
  					StrDIp.isRunning := FALSE;
  					StrDIp.isEnded := FALSE;
  					StrDIp.hasError 	:= FALSE;

  					cmd_for_Status := 0;
  					source_for_Status := source;
  					command_error_for_Status := cmd;
  				END_IF;
                                          StrDIp.inOpcCommandsDisabled:=FALSE;

                  (*cmdReset*) 2: 	StrDIp.isRunning := FALSE;
  				StrDIp.isEnded := FALSE;
  				StrDIp.hasError 	:= FALSE;
  				SignalingDi:= FALSE;
  				StrDIp.Check := FALSE;
  				cmd_for_Status := cmd;
  				source_for_Status := source;
  				command_error_for_Status := 0;
                                         StrDIp.inOpcCommandsDisabled:=FALSE;

  	(*cmd_setRemont*) 4 :	StrDIp.Remont := TRUE;
  				(*StrDIp.isRunning := FALSE;*)

  				cmd_for_Status := cmd;
  				source_for_Status := source;
  				command_error_for_Status := 0;
          (*cmd_resetRemont*) 5 : 	(*IF di.Q THEN
  					cmd_for_Status := 0;
  					source_for_Status := 0;
  					command_error_for_Status := cmd;
  				ELSE*)
  					StrDIp.Remont := FALSE;
  					(*StrDIp.isRunning := TRUE;*)

  					cmd_for_Status := cmd;
  					source_for_Status := source;
  					command_error_for_Status := 0;
  				(*END_IF;*)
  	(*cmd_setCheck*) 6 : 	StrDIp.Check := TRUE;

  				cmd_for_Status := cmd;
  				source_for_Status := source;
  				command_error_for_Status := 0;
  	END_CASE;
  	resetCmdTimer(IN := false);
  	resetCmdTimerPriznak := TRUE;
  END_IF;
  lastCmd := cmd;

  resetCmdTimer(IN := resetCmdTimerPriznak);
  IF resetCmdTimer.Q THEN
  	resetCmdTimerPriznak := FALSE;
  	source_for_Status := 0;
  	cmd_for_Status := 0;
  	command_error_for_Status := 0;
  END_IF;

  IF StrDIp.isRunning AND NOT StrDIp.Remont AND NOT StrDIp.Check THEN
  	StrDIp.Signaling := SignalingDi;
  	StrDIp.SignalingTP := _signalingTp.Q;
  ELSE
  	StrDIp.Signaling := 0;
  	StrDIp.SignalingTP := 0;
  END_IF;

  _signalingTp(in := StrDIp.Signaling, PT := T#1s);

  StrDIp.status :=  SHL(BYTE_TO_DWORD(source_for_Status), 29)
  			OR SHL(BYTE_TO_DWORD(cmd_for_Status), 26)
  			OR SHL(BYTE_TO_DWORD(command_error_for_Status), 23)
  			OR SHL(BOOL_TO_DWORD(StrDIp.OpcCommandsDisabled ), 21)
  			OR SHL(BOOL_TO_DWORD(StrDIp.Signaling), 16)
  			OR SHL(BOOL_TO_DWORD(StrDIp.RunOnStart ), 15)
  			OR SHL(BOOL_TO_DWORD(StrDIp.remont), 6)
  			OR SHL(BOOL_TO_DWORD(StrDIp.Check), 5)
  			OR SHL(BOOL_TO_DWORD(StrDIp.hasError), 4)
  			OR SHL(BOOL_TO_DWORD(StrDIp.SignalingTP), 3)
  			OR SHL(BOOL_TO_DWORD(StrDIp.CanRun), 2)
  			OR SHL(BOOL_TO_DWORD(StrDIp.isEnded), 1)
  			OR BOOL_TO_DWORD(StrDIp.isRunning);
END_FUNCTION_BLOCK

FUNCTION_BLOCK fb_DiSourceMlp
  VAR_INPUT
    arDIN : TItemDIN;
    err_mod : TItemDIN;
  END_VAR
  VAR_IN_OUT
    strDI : struct_DI;
  END_VAR
  VAR_OUTPUT
    Bounce : BOOL;
  END_VAR
  VAR
    _value : WORD;
    _reliability : BOOL;
    bitNumber : INT;
    bitNum : INT;
  END_VAR

  strDI.blConnect := TRUE;(*((UINT_TO_WORD(arDIN.wFlags) = 1472) and (UINT_TO_WORD(err_mod.wValue) = 20) and (UINT_TO_WORD(err_mod.wFlags) = 192);*)
  Bounce := (UINT_TO_WORD(arDIN.wFlags) AND 16#0020) <> 0;

  If NOT strDI.imit THEN
  _value:=UINT_TO_WORD(arDIN.wValue);

      IF strDI.blConnect THEN
            strDI.reliability:=0;
            strDI.value:=0;
  	FOR bitNumber:=0 TO 7 BY 1 DO

  		_reliability:=WORD_TO_BOOL(SHR(_value, bitNumber*2) AND 16#2);
  		strDI.reliability:=strDI.reliability OR SHL(BOOL_TO_WORD(_reliability),bitNumber);
  		IF _reliability THEN
  			strDI.value:=strDI.value OR SHL((SHR(_value, bitNumber*2) AND 16#1),bitNumber);
  		END_IF;
  	END_FOR;
      ELSE
  	strDI.reliability := 0;
      END_IF;

      FOR bitNum:=0 TO 15 BY 1 DO
  	          strDI.bits[bitNum].reliability :=WORD_TO_BOOL(SHR(strDI.reliability, bitNum) AND 16#1);
  	IF strDI.bits[bitNum].reliability THEN
  		strDI.bits[bitNum].value :=WORD_TO_BOOL(SHR(strDI.value, bitNum) AND 16#1);
                      strDI.bits[bitNum]._inversed :=NOT strDI.bits[bitNum].value;
  	END_IF;
      END_FOR;

  END_IF;
END_FUNCTION_BLOCK

FUNCTION_BLOCK fb_DiscretParametr
  VAR_IN_OUT
    StrDP : struct_DiscretParametr;
  END_VAR
  VAR
    _sunpackerCommand : fb_sunpackerCommand;
    source : BYTE;
    cmd : BYTE;
    parametr : BYTE;
    lastParametr : BYTE;
    source_for_Status : BYTE;
    cmd_for_Status : BYTE;
    command_error_for_Status : BYTE;
    resetCmdTimer : TON;
    resetCmdTimerPriznak : BOOL;
    secondTact : BOOL;
  END_VAR

  IF NOT secondTact THEN
  	StrDP.Value := StrDP.currentValue;
  	secondTact := true;
  END_IF;

  StrDP.OpcCommandsDisabled := StrDP.inOpcCommandsDisabled;

  (* ---- Если управление с ВУ заблокировано, то передаем команду из алгоритма ---- *)
  IF StrDP.inOpcCommandsDisabled THEN
  	StrDP.inCommand := StrDP.inCommand_Alg;
  ELSE (* иначе передаем команду с АРМа*)
  	StrDP.inCommand := StrDP.inCommand_ARM;
  END_IF;

  _sunpackerCommand(command := StrDP.inCommand);
  	source := _sunpackerCommand.source;
            parametr := _sunpackerCommand.parametr;
  	cmd := _sunpackerCommand.cmd;

  IF NOT StrDP.inOpcCommandsDisabled THEN
  StrDP.newValue:= BYTE_TO_UINT(parametr);
  END_IF;

  IF cmd <> 0 AND StrDP.Value <> StrDP.newValue AND (((NOT StrDP.opcCommandsDisabled) AND source > 0) OR source = 0) then
  	CASE BYTE_TO_INT(cmd) OF
  	(*cmd_ChangeValue*) 1 :
                                    StrDP.Value := StrDP.newValue;
                                    StrDP.opcCommandsDisabled:=FALSE;
  	END_CASE;
  	source_for_Status := source;
  	cmd_for_Status := cmd;
  	resetCmdTimer(IN := FALSE);
  	resetCmdTimerPriznak := TRUE;
  END_IF;

  lastParametr := parametr;

  StrDP.status := SHL(BYTE_TO_DWORD(source_for_Status), 29)
  			OR SHL(BYTE_TO_DWORD(cmd_for_Status), 26)
  			OR SHL(BYTE_TO_DWORD(command_error_for_Status), 23)
  			OR SHL(BOOL_TO_DWORD(StrDP.OpcCommandsDisabled ), 21);

  resetCmdTimer(IN := resetCmdTimerPriznak, PT := T#5S);
  IF resetCmdTimer.Q THEN
  	resetCmdTimerPriznak := FALSE;
  	source_for_Status := 0;
  	cmd_for_Status := 0;
  	command_error_for_Status := 0;
  END_IF;
END_FUNCTION_BLOCK

FUNCTION_BLOCK fb_DiscretParametr_Init
  VAR_INPUT
    data_Ini : BOOL;
    currentValue : UINT;
  END_VAR
  VAR_IN_OUT
    strDp : struct_DiscretParametr;
  END_VAR
  VAR_OUTPUT
    Init : BOOL         := FALSE;
  END_VAR

  (*****            Функциональный блок переинициализации дискретного параметра.          *****)

   Init := FALSE;

      IF data_Ini THEN                            (* Параметрам требуется переинициализация. *)
          strDp.currentValue       := currentValue;
          data_Ini:=FALSE;
          Init := TRUE;
      END_IF;
  IF Init THEN
  currentValue:=0;
  END_IF;
END_FUNCTION_BLOCK

FUNCTION_BLOCK fb_DualStateIm
  VAR_INPUT
    statOn : BOOL;
    statOff : BOOL;
  END_VAR
  VAR_IN_OUT
    StrDs : struct_DualStateIm;
  END_VAR
  VAR_INPUT
    statOn_reliability : BOOL;
    statOff_reliability : BOOL;
    inNs : TYPE_ReliableBit;
    inAccident : TYPE_ReliableBit;
    inCommand : WORD;
  END_VAR
  VAR
    _statOn : BOOL;
    _statOff : BOOL;
    lastOnStatus : BYTE;
    cmd : BYTE;
    source : BYTE;
    lastCmd : BYTE;
    source_for_Status : BYTE;
    cmd_for_Status : BYTE;
    command_error_for_Status : BYTE;
    _sunpackerCommand : fb_sunpackerCommand;
    _statusDualInput : TYPE_statusDualInput;
    _commandDualInput : TYPE_commandDualInput;
    _commandErrorTimer : BOOL;
    onInit : BOOL         := FALSE;
    resetErrorTimer : BOOL;
    _changWithoutCommand : BOOL;
    errorCMDTimer : TON;
    _errorReset : TON;
  END_VAR
  VAR_IN_OUT
    cmdOn : BOOL;
  END_VAR
  VAR_OUTPUT
    cmdOff : BOOL;
  END_VAR

  IF NOT onInit THEN
  IF StrDs.ISVALIDREF_cmdOn XOR StrDs.ISVALIDREF_cmdOff THEN
  	IF 	StrDs.ISVALIDREF_cmdOn THEN
  		lastCmd:= 2; (*baseCmdOff*)
  	ELSE
  		lastCmd:= 1; (*baseCmdOn*)
  	END_IF;
  END_IF;
  onInit:=TRUE;
  END_IF;

  (* ---- Если управление с ВУ заблокировано, то в ИМ передаем команду из алгоритма ---- *)
  IF StrDs.inOpcCommandsDisabled THEN
  	StrDs.inCommand := StrDs.inCommand_Alg;
  ELSE (* иначе передаем команду с АРМа*)
  	StrDs.inCommand := StrDs.inCommand_ARM;
  END_IF;

  (* ---- Формирование состояния механизма ---- *)

  IF (StrDs.ISVALIDREF_statOn) OR (StrDs.ISVALIDREF_statOff) THEN
  	IF (StrDs.ISVALIDREF_statOn) AND (StrDs.ISVALIDREF_statOff) THEN
  	StrDs.reliability:= statOn_reliability AND statOff_reliability;
  		_statOn  := statOn;
  		_statOff := statOff;
  	ELSIF (StrDs.ISVALIDREF_statOn) THEN
                       StrDs.reliability:= statOn_reliability;
  		_statOn  := statOn;
  		_statOff := NOT statOn;
  	ELSIF (StrDs.ISVALIDREF_statOff) THEN
  		 StrDs.reliability:= statOff_reliability;
  		_statOn  := NOT statOff;
  		_statOff :=statOff;
  	END_IF;

  	IF StrDs.reliability THEN
  		IF _statOn AND NOT _statOff 		THEN 	StrDs.onStatus := _statusDualInput.STATUS_ON;
  		ELSIF _statOff AND NOT _statOn 	THEN 	StrDs.onStatus := _statusDualInput.Status_OFF;
  		ELSIF NOT _statOn AND NOT _statOff 	THEN 	StrDs.onStatus := _statusDualInput.STATUS_TRANSITIONAL;
  		ELSE					StrDs.onStatus := _statusDualInput.STATUS_ERROR;
                      END_IF;

  	ELSE
  		StrDs.onStatus := _statusDualInput.STATUS_NOTDEFINED;

  	END_IF;
  ELSE
  	CASE BYTE_TO_INT(lastCmd) OF
  		(*baseCmdOn*) 1: StrDs.onStatus  := _statusDualInput.STATUS_ON;
  		(*baseCmdOff*) 2: StrDs.onStatus  := _statusDualInput.STATUS_OFF;

  	ELSE
  		 StrDs.onStatus := _statusDualInput.STATUS_NOTDEFINED;

  	END_CASE;
  END_IF;

  (* ---- Формирование признака сдвига ---- *)
  StrDs.sdvig  := FALSE;
  IF StrDs.ISVALIDREF_cmdOn OR StrDs.ISVALIDREF_cmdOff THEN
  	IF cmd = 0 THEN
  		IF (lastOnStatus <> StrDs.onStatus AND
  		(StrDs.onStatus <> _statusDualInput.STATUS_NOTDEFINED AND StrDs.onStatus <> _statusDualInput.STATUS_ERROR) AND
  		(lastOnStatus <> _statusDualInput.STATUS_NOTDEFINED AND lastOnStatus <> _statusDualInput.STATUS_ERROR)) THEN
  			StrDs.sdvig   := TRUE;
  		END_IF;
  	END_IF;
  END_IF;
  lastOnStatus := StrDs.onStatus;

  StrDs.Accident := inAccident.value AND inAccident.reliability;
  StrDs.Ns := inNs.value AND inNs.reliability;
  StrDs.OpcCommandsDisabled := StrDs.inOpcCommandsDisabled;

  (* ---- Распаковка команды ---- *)
  _sunpackerCommand(command := StrDs.inCommand);
  	cmd := _sunpackerCommand.cmd;
  	source := _sunpackerCommand.source;

  (* ---- Обработка команды ---- *)
  IF cmd <> 0 AND lastCmd <> cmd and (((NOT StrDs.opcCommandsDisabled) AND source > 0) OR source = 0) then
  	CASE BYTE_TO_INT(cmd) OF
  	(*cmd_open*) 1 :
  			IF  StrDs.ISVALIDREF_cmdOn THEN StrDs.CmdOn := TRUE;
  				IF StrDs.ISVALIDREF_cmdOff THEN StrDs.CmdOff := FALSE; END_IF;
  			ELSIF  StrDs.ISVALIDREF_cmdOff THEN StrDs.CmdOff := FALSE;  END_IF;
  			errorCMDTimer(IN := false);
  			_commandErrorTimer := true;
  			StrDs.lastCmdIsOn := true;
  	(*cmd_close*) 2 :
  			IF StrDs.ISVALIDREF_cmdOff THEN StrDs.CmdOff := TRUE;
  				IF StrDs.ISVALIDREF_cmdOn THEN StrDs.CmdOn := FALSE; END_IF;
  			ELSIF StrDs.ISVALIDREF_cmdOn THEN StrDs.CmdOn := FALSE; END_IF;
  			errorCMDTimer(IN := false);
  			_commandErrorTimer := true;
  			StrDs.lastCmdIsOn := false;
  	(*cmd_reset*) 3 :    IF StrDs.ISVALIDREF_statOn OR StrDs.ISVALIDREF_statOff THEN
  			StrDs.CmdOn := FALSE;
  			StrDs.CmdOff := FALSE;
                                lastCmd :=0;
  			_commandErrorTimer := false;
  			StrDs.lastCmdIsOn := false;
                                END_IF;
  	END_CASE;
  	source_for_Status := source;
  	cmd_for_Status := cmd;
  	command_error_for_Status := 0;
  END_IF;

  lastCmd := cmd;
  errorCMDTimer(In := _commandErrorTimer, PT :=T#10s);

  (* ---- алгоритм  для команды ВКЛючить ---- *)
  IF (StrDs.onStatus = _statusDualInput.STATUS_ON) and (lastCmd = _commandDualInput.CMD_ON) then
  	IF StrDs.ISVALIDREF_cmdOn AND StrDs.ISVALIDREF_cmdOff then  StrDs.cmdOn := false; END_IF;

  	 errorCMDTimer(In := false);
  	 _commandErrorTimer := false;
  	 cmd_for_Status := 0;
  	 source_for_Status := 0;
  END_IF;

  (* ---- off ---- *)
  IF (StrDs.onStatus = _statusDualInput.STATUS_OFF) and (lastCmd = _commandDualInput.CMD_OFF) then
  	IF StrDs.ISVALIDREF_cmdOn AND StrDs.ISVALIDREF_cmdOff then  StrDs.cmdOff := false; END_IF;

  	 errorCMDTimer(In := false);
  	 _commandErrorTimer := false;
  	 cmd_for_Status := 0;
  	 source_for_Status := 0;
  END_IF;

  (* ---- ошибка исполнения команды ---- *)
  if errorCMDTimer.Q and (cmd_for_Status <> 0) then
  	command_error_for_Status :=  cmd_for_Status;
  	_commandErrorTimer := false;
  	StrDs.CmdOn := false;
  	StrDs.CmdOff := false;
  	lastCmd := 0;
  end_if;

  (* ---- сброс ошибки команды ---- *)
  StrDs.CommandFault := command_error_for_Status <> 0;
  _errorReset(IN := command_error_for_Status <> 0, PT := T#15S);
  IF _errorReset.Q THEN
  	cmd_for_Status := 0;
  	source_for_Status := 0;
  	command_error_for_Status := 0;
  END_IF;

  cmdOn := StrDs.cmdOn;
  cmdOff:= StrDs.cmdOff;

  (* ---- формирование зашифрованного статуса для АРМа ---- *)
  StrDs.status := shl(BYTE_TO_DWORD(source_for_Status), 29)
  		OR shl(BYTE_TO_DWORD(cmd_for_Status), 26)
  		OR shl(BYTE_TO_DWORD(command_error_for_Status), 23)
  		OR shl(bool_to_DWORD(StrDs.sdvig), 22)
  		OR shl(bool_to_DWORD(StrDs.OpcCommandsDisabled), 21)
  		OR shl(BOOL_TO_DWORD(StrDs.Ns), 4)
                  	OR shl(BOOL_TO_DWORD(StrDs.Accident ),3)
  		OR BYTE_TO_DWORD(StrDs.onStatus);
END_FUNCTION_BLOCK

FUNCTION_BLOCK fb_Kran
  VAR_INPUT
    statOn : BOOL;
    statOff : BOOL;
    statOn_reliability : BOOL;
    statOff_reliability : BOOL;
  END_VAR
  VAR_IN_OUT
    strKr : struct_Kran;
  END_VAR
  VAR_INPUT
    inNs : TYPE_ReliableBit;
    inAccident : TYPE_ReliableBit;
    inAuto : TYPE_ReliableBit;
    inManual : TYPE_ReliableBit;
    inLocal : TYPE_ReliableBit;
    inDistance : TYPE_ReliableBit;
    inErrorPowerOff : TYPE_ReliableBit;
    inErrorBlock : TYPE_ReliableBit;
    inSo : TYPE_ReliableBit;
    inSz : TYPE_ReliableBit;
    inDp : TYPE_ReliableBit;
  END_VAR
  VAR
    _reliability : BOOL;
    onInit : BOOL         := FALSE;
    _statOn : BOOL;
    _statOff : BOOL;
    lastOnStatus : BYTE;
    cmd : BYTE;
    source : BYTE;
    lastCmd : BYTE;
    source_for_Status : BYTE;
    cmd_for_Status : BYTE;
    command_error_for_Status : BYTE;
    _sunpackerCommand : fb_sunpackerCommand;
    _statusDualInput : TYPE_statusDualInput;
    _commandDualInput : TYPE_commandDualInput;
    _commandErrorTimer : BOOL;
    resetErrorTimer : BOOL;
    _changWithoutCommand : BOOL;
    BlockedOpenControl : BOOL;
    errorCMDTimer : TON;
    _errorReset : TON;
    continueHoldCommandTimer : TON;
    outputsSets : TOF;
    dP_Trig : R_TRIG;
    dP_Trig_reliability : R_TRIG;
    resetBlockedOpenControl_Trig : R_TRIG;
  END_VAR
  VAR_IN_OUT
    cmdOn : BOOL;
    cmdOff : BOOL;
  END_VAR

  IF NOT onInit THEN
  IF strKr.ISVALIDREF_cmdOn XOR strKr.ISVALIDREF_cmdOff THEN
  	IF 	strKr.ISVALIDREF_cmdOn THEN
  		lastCmd:= 2; (*baseCmdOff*)
  	ELSE
  		lastCmd:= 1; (*baseCmdOn*)
  	END_IF;
  END_IF;
  onInit:=TRUE;
  END_IF;

  (* ---- Если управление с ВУ заблокировано, то в ИМ передаем команду из алгоритма ---- *)
  IF strKr.inOpcCommandsDisabled THEN
  	strKr.inCommand := strKr.inCommand_Alg;
  ELSE (* иначе передаем команду с АРМа*)
  	strKr.inCommand := strKr.inCommand_ARM;
  END_IF;

  (* ---- Формирование состояния механизма ---- *)

  IF (strKr.ISVALIDREF_statOn) OR (strKr.ISVALIDREF_statOff) THEN
  	IF (strKr.ISVALIDREF_statOn) AND (strKr.ISVALIDREF_statOff) THEN
  	_reliability:= statOn_reliability AND statOff_reliability;
  		_statOn  := statOn;
  		_statOff := statOff;
  	ELSIF (strKr.ISVALIDREF_statOn) THEN
                       _reliability:= statOn_reliability;
  		_statOn  := statOn;
  		_statOff := NOT statOn;
  	ELSIF (strKr.ISVALIDREF_statOff) THEN
  		 _reliability:= statOff_reliability;
  		_statOn  := NOT statOff;
  		_statOff :=statOff;
  	END_IF;

  	IF _reliability THEN
  		IF _statOn AND NOT _statOff 		THEN 	strKr.onStatus := _statusDualInput.STATUS_ON;
  		ELSIF _statOff AND NOT _statOn 	THEN 	strKr.onStatus := _statusDualInput.Status_OFF;
  		ELSIF NOT _statOn AND NOT _statOff 	THEN 	strKr.onStatus := _statusDualInput.STATUS_TRANSITIONAL;
  		ELSE					strKr.onStatus := _statusDualInput.STATUS_ERROR;
                      END_IF;

  	ELSE
  		strKr.onStatus := _statusDualInput.STATUS_NOTDEFINED;

  	END_IF;
  ELSE
  	CASE BYTE_TO_INT(lastCmd) OF
  		(*baseCmdOn*)  1: strKr.onStatus  := _statusDualInput.STATUS_ON;
  		(*baseCmdOff*) 2: strKr.onStatus  := _statusDualInput.STATUS_OFF;

  	ELSE
  		 strKr.onStatus := _statusDualInput.STATUS_NOTDEFINED;

  	END_CASE;
  END_IF;

  strKr.Accident := inAccident.value AND inAccident.reliability;
  strKr.Ns := inNs.value AND inNs.reliability;
  strKr.Auto := inAuto.value AND inAuto.reliability;
  strKr.Manual := inManual.value AND inManual.reliability;
  strKr.Local := inLocal.value AND inLocal.reliability;
  strKr.Distance := inDistance.value AND inDistance.reliability;
  strKr.ErrorPowerOff := inErrorPowerOff.value AND inErrorPowerOff.reliability;
  strKr.ErrorBlock := inErrorBlock.value AND inErrorBlock.reliability;
  strKr.OpcCommandsDisabled := strKr.inOpcCommandsDisabled;

  (* ---- Формирование признака блокировки Открытия крана по высокому давлению ---- *)
  	IF strKr.ISVALIDREF_inDp THEN

  		strKr.Dp := inDp.value AND inDp.reliability;

  		dP_Trig(CLK := strKr.Dp );
  		dP_Trig_reliability(CLK :=NOT inDp.reliability);

  		IF dP_Trig.Q OR dP_Trig_reliability.Q THEN
  			BlockedOpenControl := TRUE;
  		END_IF;
  		(* ---- автоматический сброс *)
  		resetBlockedOpenControl_Trig(CLK := (NOT inDp.value) AND inDp.reliability);
  		IF resetBlockedOpenControl_Trig.Q THEN
  			BlockedOpenControl := FALSE;
  		END_IF;
  	ELSE
  		strKr.Dp  := FALSE;
  		BlockedOpenControl := FALSE;
  	END_IF;

  (* ---- Формирование признака сдвига ---- *)
  strKr.sdvig  := FALSE;
  IF (strKr.ISVALIDREF_cmdOn OR strKr.ISVALIDREF_cmdOff) AND NOT strKr.Local THEN
  	IF cmd = 0 THEN
  		IF (lastOnStatus <> strKr.onStatus AND
  		(strKr.onStatus <> _statusDualInput.STATUS_NOTDEFINED AND strKr.onStatus <> _statusDualInput.STATUS_ERROR) AND
  		(lastOnStatus <> _statusDualInput.STATUS_NOTDEFINED AND lastOnStatus <> _statusDualInput.STATUS_ERROR)) THEN
  			strKr.sdvig   := TRUE;
  		END_IF;
  	END_IF;
  END_IF;
  lastOnStatus := strKr.onStatus;

  (* ---- Распаковка команды ---- *)
  _sunpackerCommand(command := strKr.inCommand);
  	cmd := _sunpackerCommand.cmd;
  	source := _sunpackerCommand.source;

  (* ---- Обработка команды ---- *)
  IF cmd <> 0 AND lastCmd <> cmd and (((NOT strKr.opcCommandsDisabled) AND source > 0) OR source = 0) then
  	CASE BYTE_TO_INT(cmd) OF
  	(*cmd_open*) 1 :
  			IF NOT BlockedOpenControl THEN
                                IF  strKr.ISVALIDREF_cmdOn THEN strKr.CmdOn := TRUE;
  				IF strKr.ISVALIDREF_cmdOff THEN strKr.CmdOff := FALSE; END_IF;
  			ELSIF  strKr.ISVALIDREF_cmdOff THEN strKr.CmdOff := FALSE;  END_IF;
  			errorCMDTimer(IN := false);

  			_commandErrorTimer := true;
  			strKr.lastCmdIsOn := true;
                                END_IF;
  	(*cmd_close*) 2 :
  			IF strKr.ISVALIDREF_cmdOff THEN strKr.CmdOff := TRUE;
  				IF strKr.ISVALIDREF_cmdOn THEN strKr.CmdOn := FALSE; END_IF;
  			ELSIF strKr.ISVALIDREF_cmdOn THEN strKr.CmdOn := FALSE; END_IF;
  			errorCMDTimer(IN := false);

  			_commandErrorTimer := true;
  			strKr.lastCmdIsOn := false;
  	(*cmd_reset*) 3 :   IF (strKr.ISVALIDREF_statOn) OR (strKr.ISVALIDREF_statOff) THEN
  			strKr.CmdOn := FALSE;
  			strKr.CmdOff := FALSE;
                                lastCmd := 0;
  			_commandErrorTimer := false;
  			strKr.lastCmdIsOn := false;
                                END_IF;

  	END_CASE;
  	source_for_Status := source;
  	cmd_for_Status := cmd;
  	command_error_for_Status := 0;
  END_IF;
  lastCmd := cmd;
